// ---- GlobalTextList.TcGTLO
TEXTLIST GlobalTextList
  577 = ''
  578 = '%.1f'
  1916 = '%.1f '
  272 = '%.1f s'
  1255 = '%.2f'
  522 = '%.2f '
  324 = '%d'
  534 = '%i'
  168 = '%s'
  467 = '+'
  2312 = '+/-%.1f '
  462 = '+/-%.2f '
  1236 = '+/-%.f '
  759 = '-'
  43 = '1. Ben chặn hũ trên (s)' | vn: '1. Ben chặn hũ trên (s)' | eng: '1. Upper cylinder blocks jar (s)'
  1848 = '1. Ben dập nắp' | vn: '1. Ben dập nắp' | eng: '1. Cylinder presses lid'
  610 = '1. Ben dập nắp (s)' | vn: '1. Ben dập nắp (s)' | eng: '1. Cylinder presses lid (s)'
  2468 = '1. Ben hút, thả nắp' | vn: '1. Ben hút, thả nắp' | eng: '1. Cylinder sucks/release lid'
  1761 = '1. Ben hút/thả nắp (s)' | vn: '1. Ben hút/thả nắp (s)' | eng: '1. Cylinder sucks/release lid (s)'
  1520 = '1. Ben lược vào/ra' | vn: '1. Ben lược vào/ra' | eng: '1. Comb cylinder moves in/out'
  194 = '1. Ben lược vào/ra (s)' | vn: '1. Ben lược vào/ra (s)' | eng: '1. Comb cylinder moves in/out (s)'
  2358 = '1. Motor đảo thức ăn (Hz)' | vn: '1. Động cơ đảo thức ăn (Hz)' | eng: '1. Food Agitator motor (Hz)'
  2242 = '1. Phễu rung (Hz)' | vn: '1. Phễu rung (Hz)' | eng: '1. Vibrating funnel (Hz)'
  1784 = '1. Thời gian cân sâu (s)' | vn: '1. Thời gian cân sâu (s)' | eng: '1. Time for weighting larvae (s)'
  368 = '1. Thời gian cân thức ăn (s)' | vn: '1. Thời gian cân thức ăn (s)' | eng: '1. Time for weighting food (s)'
  621 = '1.Ben chặn hũ trên' | vn: '1. Ben chặn hũ trên' | eng: '1. The upper cylinder blocks the jar'
  1429 = '1.Khối lượng (g)' | vn: '1. Khối lượng (g)' | eng: '1. The mass (g)'
  758 = '1.Khối lượng yêu cầu (g)' | vn: '1. Khối lượng yêu cầu (g)' | eng: '1. The desire mass (g)'
  1103 = '1.Số Shoot' | vn: '1. Số Shoot' | eng: '1. Shoot number'
  1518 = '1/2'
  870 = '10. Khoảng trễ (s)' | vn: '10. Khoảng trễ (s)' | eng: '10. Delay (s)'
  2444 = '11. Tốc độ băng tải đầu ra (Hz)' | vn: '11. Tốc độ băng tải đầu ra (Hz)' | eng: '11. Speed of output conveyor (Hz)'
  3265 = '11. Tốc độ đảo thức ăn (Hz)' | vn: '11. Tốc độ đảo thức ăn (Hz)' | eng: '11. Speed of agitator motor (Hz)'
  3571 = '11. Tốc độ động cơ đảo (Hz)' | vn: '11. Tốc độ động cơ đảo (Hz)' | eng: '11. Speed of agitator motor (Hz)'
  254 = '2. Ben chặn hũ dưới (s)' | vn: '2. Ben chặn hũ dưới (s)' | eng: '2. Lower cylinder blocks jar (s)'
  85 = '2. Ben chặn nắp (s)' | vn: '2. Ben chặn nắp (s)' | eng: '2. Cylinder blocks lid (s)'
  2129 = '2. Ben chặn nắp trên ray' | vn: '2. Ben chặn nắp trên ray' | eng: '2. Cylinder blocks lid in rail'
  4542 = '2. Ben chặn sâu' | vn: '2. Ben chặn sâu ' | eng: '2. Cylinder blocks larvae'
  89 = '2. Ben di chuyển lược' | vn: '2. Ben di chuyển lược' | eng: '2. Cylinder moves comb'
  1937 = '2. Ben kẹp hũ (s)' | vn: '2. Ben kẹp hũ (s)' | eng: '2. Cylinder clamp jar (s)'
  1481 = '2. Khoảng trễ ben dập nắp rút về (s)' | vn: '2. Thời gian ben dập nắp rút về (s)' | eng: '2. Time for cylinder pressing lid retract (s)'
  204 = '2. Motor chia thức ăn (rpm)' | vn: '2. Động cơ chia thức ăn (rpm)' | eng: '2. Food dispenser motor (rpm)'
  588 = '2. Sai số (%)' | vn: '2. Sai số (%)' | eng: '2. Deviation (%)'
  863 = '2. Sai số cho phép (%)' | vn: '2. Sai số cho phép (%)' | eng: '2. Allowable deviation (%)'
  4394 = '2. Thời gian ben dập nắp rút về (s)' | vn: '2. Thời gian ben dập nắp rút về (s)' | eng: '2. Time for cylinder pressing lid retract (s)'
  2355 = '2. Thời gian ổn định hũ sâu (s)' | vn: '2. Thời gian ổn định hũ sâu (s)' | eng: '2. Time to stabilize the larvae jar (s)'
  4032 = '2. Thời gian ổn định hũ thức ăn (s)' | vn: '2. Thời gian ổn định hũ thức ăn (s)' | eng: '2. Time to stabilize the food jar (s)'
  311 = '2.Ben chặn hũ dưới' | vn: '2. Ben chặn hũ dưới' | eng: '2. The lower cylinder blocks the jar'
  3026 = '2/2'
  98 = '3. Ben chặn sâu (s)' | vn: '3. Ben chặn sâu (s)' | eng: '3. Cylinder blocks larvae (s)'
  198 = '3. Ben di chuyển lược (s)' | vn: '3. Ben di chuyển lược (s)' | eng: '3. Cylinder moves comb (s)'
  1881 = '3. Ben kẹp hũ, đối diện lược' | vn: '3. Ben kẹp hũ, đối diện lược' | eng: '3. Cylinder clamp the jar (s)'
  779 = '3. Kiểm tra hết hũ (s)' | vn: '3. Kiểm tra hết hũ (s)' | eng: '3. The jar is getting low (s)'
  1590 = '3. Kiểm tra hết nắp (s)' | vn: '3. Kiểm tra hết nắp (s)' | eng: '3. The lid is getting low (s)'
  1960 = '3. Thời gian đảo chiều động cơ trộn thức ăn (s)' | vn: '3. Thời gian đảo chiều động cơ trộn thức ăn (s)' | eng: '3. Timer for reversing agitator motor (s)'
  952 = '3. Tốc độ cấp I (Hz)' | vn: '3. Tốc độ cấp I (Hz)' | eng: '3. The velocity (Hz)'
  455 = '3. Tốc độ cấp I (rpm)' | vn: '3. Tốc độ cấp I (rpm)' | eng: '3. The velocity I (rpm)'
  3651 = '3. Tốc độ I (Hz)' | vn: '3. Tốc độ I (Hz)' | eng: '3. The velocity I (Hz)'
  1182 = '3. Tốc độ I (rpm)' | vn: '3. Tốc độ I (rpm)' | eng: '3. The velocity I (rpm)'
  3921 = '3. Van hút nắp' | vn: '3. Van hút nắp' | eng: '3. Valve sucks lid '
  740 = '3.Ben hút/thả hũ' | vn: '3. Ben hút/thả hũ' | eng: '3. Cylinder sucks/release jar'
  594 = '4. Kiểm tra hút được nắp (s)' | vn: '4. Kiểm tra hút được nắp (s)' | eng: '4. The lid is suctioned (s)'
  413 = '4. Kiểm tra hết sâu (s)' | vn: '4. Kiểm tra hết sâu (s)' | eng: '4. Check running out of larvae (s)'
  1166 = '4. Kiểm tra kẹt hũ (s)' | vn: '4. Kiểm tra kẹt hũ (s)' | eng: '4. The jar is stucked (s)'
  118 = '4. Thời gian đảo chiều động cơ chia thức ăn (s)' | vn: '4. Thời gian đảo chiều động cơ chia thức ăn (s)' | eng: '4. Timer for reversing (s)'
  4404 = '4. Tốc độ cấp II (Hz)' | vn: '4. Tốc độ cấp II (Hz)' | eng: '4. The velocity I (Hz)'
  297 = '4. Tốc độ cấp II (rpm)' | vn: '4. Tốc độ cấp II (rpm)' | eng: '4. The velocity II (rpm)'
  1764 = '4. Tốc độ II (Hz)' | vn: '4. Tốc độ II (Hz)' | eng: '4. The velocity II (Hz)'
  344 = '4. Tốc độ II (rpm)' | vn: '4. Tốc độ II (rpm)' | eng: '4. The velocity II (rpm)'
  86 = '4. Van hút định vị hũ' | vn: '4. Van hút định vị hũ' | eng: '4. Suction valve locates the jar'
  2844 = '5. Ben chặn hũ trên đẩy ra (s)' | vn: '5. Ben chặn hũ trên đẩy ra (s)' | eng: '5. Upper clinder blocks jar extend (s)'
  2498 = '5. Kiểm tra hết thức ăn (s)' | vn: '5, Kiểm tra hết thức ăn (s)' | eng: '5. Check running out of food (s)'
  2430 = '5. Ngắt hút (s)' | vn: '5. Ngắt hút (s)' | eng: '5. Shut off suction (s)'
  3883 = '5. Tốc độ cấp III (Hz)' | vn: '5. Tốc độ cấp III (Hz)' | eng: '5. The velocity III (Hz)'
  1037 = '5. Tốc độ cấp III (rpm)' | vn: '5. Tốc độ cấp III (rpm)' | eng: '5. The velocity III (rpm)'
  4207 = '5. Tốc độ III (Hz)' | vn: '5. Tốc độ III (Hz)' | eng: '5. The velocity III (Hz)'
  353 = '5. Tốc độ III (rpm)' | vn: '5. Tốc độ III (rpm)' | eng: '5. The velocity III (rpm)'
  2962 = '6. Ben hút/thả hũ (s)' | vn: '6. Ben hút/thả hũ (s)' | eng: '6. Cylinder sucks/releases jar (s)'
  2859 = '6. Ben hút/thả hũ(s)' | vn: '6. Ben hút/thả hũ (s)' | eng: '6. Cylinder sucks/releases jar (s)'
  657 = '6. Chuyển I - II (%)' | vn: '6. Chuyển I - II (%)' | eng: '6. Change I - II (%)'
  18 = '6. Vị trí chuyển cấp I - II (%)' | vn: '6. Vị trí chuyển cấp I - II (%)' | eng: '6. Postion change speed I - II (%)'
  1654 = '7. Ben hút/thả hũ rút về (s)' | vn: '7. Ben hút/thả hũ rút về (s)' | eng: '7. Cylinder sucks/releases jar retract (s)'
  865 = '7. Chuyển II - III (%)' | vn: '7. Chuyển II - III (%)' | eng: '7. Change II - III (%)'
  564 = '7. Vị trí chuyển cấp II - III (%)' | vn: '7. Vị trí chuyển cấp II - III (%)' | eng: '7. Position change speed II - III (%)'
  965 = '8. Ngắt hút (s)' | vn: '8. Ngắt hút (s)' | eng: '8. Stop suction (s)'
  677 = '8. Tải trọng tối đa (g)' | vn: '8. Tải trọng tối đa (g)' | eng: '8. Maximum payload (g)'
  1330 = '9. Vị trí dừng (%)' | vn: '9. Vị trí dừng (%)' | eng: '9. Halt position (%)'
  1341 = '9.Kích hút (s)' | vn: '9. Kích hút (s)' | eng: '9. Suction (s)'
  2827 = 'Bypass cửa' | vn: 'Bypass cửa' | eng: 'Bypass door'
  1689 = 'Bypass Nắp' | vn: 'Bypass Nắp' | eng: 'Bypass lid'
  1003 = 'Bypass Sâu' | vn: 'Bypass Sâu' | eng: 'Bypass larvae'
  207 = 'Bypass Thức ăn' | vn: 'Bypass Thức ăn' | eng: 'Bypass food'
  642 = 'Bạn có muốn xóa không?' | vn: 'Bạn có muốn xóa không?' | eng: 'Do you want to delete?'
  917 = 'Chạy' | vn: 'Chạy' | eng: 'Run'
  137 = 'Clear' | vn: 'Xóa' | eng: 'Clear'
  352 = 'Cài đặt' | vn: 'Cài đặt' | eng: 'Setting'
  503 = 'Có' | vn: 'Có' | eng: 'Yes'
  689 = 'Cụm cân sâu' | vn: 'Cụm cân sâu' | eng: 'Weighing larvae'
  775 = 'Cụm cấp hũ' | vn: 'Cụm cấp hũ' | eng: 'Jar supply'
  129 = 'Cụm cấp nắp' | vn: 'Cụm cấp nắp' | eng: 'Lid supply'
  838 = 'Cụm cấp thức ăn' | vn: 'Cụm cấp thức ăn' | eng: 'Food supply'
  454 = 'Cụm dập nắp' | vn: 'Cụm dập nắp' | eng: 'Pressing lid'
  80 = 'Cụm transfer' | vn: 'Cụm transfer' | eng: 'Transfer'
  1210 = 'DELAY LINE 1' | vn: 'THỜI GIAN TRẠM 1' | eng: 'TIMER LINE 1'
  1442 = 'DELAY LINE 2' | vn: 'THỜI GIAN TRẠM 2' | eng: 'TIMER LINE 2'
  61 = 'Describe'
  236 = 'Dừng' | vn: 'Dừng' | eng: 'Stop'
  643 = 'Dừng hút' | vn: 'Dừng hút' | eng: 'Stop suction'
  781 = 'Engineer'
  196 = 'Hút' | vn: 'Hút' | eng: 'Suck'
  2112 = 'Hết ca' | vn: 'Hết ca' | eng: 'End shift'
  1181 = 'ID' | vn: 'ID' | eng: 'ID'
  836 = 'INPUT' | vn: 'NGÕ VÀO' | eng: 'INPUT'
  184 = 'Không' | vn: 'Không' | eng: 'No'
  640 = 'Khối lượng cốc (g)' | vn: 'Khối lượng cốc (g)' | eng: 'Mass of cup (g)'
  523 = 'Khối lượng sâu (g)' | vn: 'Khối lượng sâu (g)' | eng: 'Mass of larvae (g)'
  474 = 'Khối lượng thức ăn (g)' | vn: 'Khối lượng thức ăn (g)' | eng: 'Mass of food (g)'
  1680 = 'LINE 1' | vn: 'TRẠM 1' | eng: 'LINE 1'
  1088 = 'LINE 2' | vn: 'TRẠM 2' | eng: 'LINE 2'
  849 = 'Lưu' | vn: 'Lưu' | eng: 'Save'
  1378 = 'Lựa chọn của bạn' | vn: 'Lựa chọn của bạn' | eng: 'Your choice'
  257 = 'MÀN HÌNH CHÍNH LINE 1' | vn: 'MÀN HÌNH CHÍNH TRẠM 1' | eng: 'MAIN LINE 1 SCREEN'
  4 = 'MÀN HÌNH CHÍNH LINE 2' | vn: 'MÀN HÌNH CHÍNH TRẠM 2' | eng: 'MAIN LINE 2 SCREEN'
  1168 = 'MÀN HÌNH CHẠY TAY LINE 1' | vn: 'MÀN HÌNH CHẠY TAY TRẠM 1' | eng: 'MANUAL LINE 1 SCREEN'
  762 = 'MÀN HÌNH CHẠY TAY LINE 2' | vn: 'MÀN HÌNH CHẠY TAY TRẠM 2' | eng: 'MANUAL LINE 2 SCREEN'
  1368 = 'MÀN HÌNH CÀI KHOẢNG TRỄ LINE 1' | vn: 'MÀN HÌNH CÀI KHOẢNG TRỄ TRẠM 1' | eng: 'SETTING DELAYS LINE 1'
  1237 = 'MÀN HÌNH CÀI KHOẢNG TRỄ LINE 2' | vn: 'MÀN HÌNH CÀI KHOẢNG TRỄ TRẠM 2' | eng: 'SETTING DELAYS LINE 2'
  386 = 'MÀN HÌNH CÀI ĐẶT LINE 1' | vn: 'MÀN HÌNH CÀI ĐẶT TRẠM 1' | eng: 'SETTINGS LINE 1 SCREEN'
  1892 = 'MÀN HÌNH CÀI ĐẶT LINE 2' | vn: 'MÀN HÌNH CÀI ĐẶT TRẠM 2' | eng: 'SETTINGS LINE 2 SCREEN'
  786 = 'MÀN HÌNH IO LINE 1' | vn: 'MÀN HÌNH IO TRẠM 1' | eng: 'IO LINE 1 SCREEN'
  798 = 'MÀN HÌNH IO LINE 2' | vn: 'MÀN HÌNH IO TRẠM 2' | eng: 'IO LINE 2 SCREEN'
  833 = 'MÀN HÌNH LƯU THÔNG SỐ LINE 1' | vn: 'MÀN HÌNH LƯU THÔNG SỐ TRẠM 1' | eng: 'PARAMETERS STORAGE LINE 1'
  1067 = 'MÀN HÌNH LƯU THÔNG SỐ LINE 2' | vn: 'MÀN HÌNH LƯU THÔNG SỐ TRẠM 2' | eng: 'PARAMETERS STORAGE LINE 2'
  4017 = 'MÀN HÌNH LỖI TRẠM 1' | vn: 'MÀN HÌNH LỖI TRẠM 1' | eng: 'ALARM SCREEN LINE 1'
  1028 = 'MÀN HÌNH LỖI TRẠM 2' | vn: 'MÀN HÌNH LỖI TRẠM 2' | eng: 'ALARM SCREEN LINE 2'
  1780 = 'MÀN HÌNH THÔNG SỐ TRẠM 1' | vn: 'MÀN HÌNH THÔNG SỐ TRẠM 1' | eng: 'PARAMETERS SCREEN LINE 1'
  1857 = 'MÀN HÌNH THÔNG SỐ TRẠM 2' | vn: 'MÀN HÌNH THÔNG SỐ TRẠM 2' | eng: 'PARAMETERS SCREEN LINE 2'
  1188 = 'Mô tả' | vn: 'Mô tả' | eng: 'Description'
  1449 = 'Ngược' | vn: 'Ngược' | eng: 'Reverse'
  777 = 'None'
  1079 = 'Năng suất (cup/h)' | vn: 'Năng suất(cốc/h)\t\t' | eng: 'Product(cup/h)'
  669 = 'Nạp' | vn: 'Nạp' | eng: 'Load'
  784 = 'Operator'
  219 = 'OUTPUT' | vn: 'NGÕ RA' | eng: 'OUTPUT'
  1453 = 'PARAMETER' | vn: 'THÔNG SỐ' | eng: 'PARAMETER'
  886 = 'Rút về' | vn: 'Rút về' | eng: 'Retract'
  139 = 'Sai số sâu (%)' | vn: 'Sai số sâu (%)' | eng: 'Deviation of larvae (%)'
  625 = 'Sai số thức ăn (%)' | vn: 'Sai số thức ăn (%)' | eng: 'Deviation of food (%)'
  478 = 'START' | vn: 'Bắt đầu' | eng: 'Start'
  3882 = 'Start page' | vn: 'Start page' | eng: 'Start page'
  440 = 'Status'
  12 = 'STOP' | vn: 'Dừng' | eng: 'Stop'
  62 = 'Sâu' | vn: 'Sâu' | eng: 'Larva'
  587 = 'SÂU' | vn: 'Sâu' | eng: 'Larva'
  909 = 'TG cân sâu' | vn: 'TG cân sâu' | eng: 'Time of weight larvae'
  2214 = 'TG cân thức ăn' | vn: 'TG cân thức ăn' | eng: 'Time of weight food'
  2059 = 'Thuận' | vn: 'Thuận' | eng: 'Forward'
  1204 = 'Thời gian' | vn: 'Thời gian' | eng: 'Time'
  1876 = 'Thời gian (s)' | vn: 'Thời gian (s)' | eng: 'Time (s)'
  294 = 'Thức ăn' | vn: 'Thức ăn' | eng: 'Food'
  513 = 'THỨC ĂN' | vn: 'Thức ăn' | eng: 'Food'
  877 = 'Thực tế' | vn: 'Thực tế' | eng: 'Actual'
  48 = 'Time'
  1196 = 'Trạng thái' | vn: 'Trạng thái' | eng: 'Status'
  771 = 'Trạng thái hoạt động' | vn: 'Trạng thái hoạt động' | eng: 'Operation status'
  1711 = 'Trộn' | vn: 'Trộn' | eng: 'Mix'
  2142 = 'Tạm dừng' | vn: 'Tạm dừng' | eng: 'Pause'
  2305 = 'Tốc độ (g/s)' | vn: 'Tốc độ (g/s)' | eng: 'Velocity (g/s)'
  754 = 'Tổng khối lượng (g)' | vn: 'Tổng khối lượng (g)' | eng: 'Mass total (g)'
  1399 = 'Tổng số cốc đã cân' | vn: 'Tổng số cốc đã cân' | eng: 'Total cups weighted'
  1621 = 'U1I1-1. Nút Start' | vn: 'U1I1-1. Nút Start' | eng: 'U1I1-1. Start button'
  3076 = 'U1I1-2. Nút Stop' | vn: 'U1I1-2. Nút Stop' | eng: 'U1I1-2. Stop button'
  536 = 'U1I1-3. Nút Reset' | vn: 'U1I1-3. Nút Reset' | eng: 'U1I1-3. Rest button'
  3249 = 'U1I2-4. Cảm biến báo thiếu hũ' | vn: 'U1I2-4. Cảm biến báo thiếu hũ' | eng: 'U1I2-4. Sensor detecting jar is getting low'
  2058 = 'U1I2-5. Cảm biến rút về của ben chặn hũ trên' | vn: 'U1I2-5. Cảm biến rút về của ben chặn hũ trên' | eng: 'U1I2-5. Retract sensor of upper cylinder'
  1695 = 'U1I2-6. Cảm biến rút về của ben chặn hũ dưới' | vn: 'U1I2-6. Cảm biến rút về của ben chặn hũ dưới' | eng: 'U1I2-6. Retract sensor of lower cylinder'
  3389 = 'U1I2-7. Cảm biến đẩy ra của ben chặn hũ dưới' | vn: 'U1I2-7. Cảm biến đẩy ra của ben chặn hũ dưới' | eng: 'U1I2-7. Extend sensor of upper cylinder'
  71 = 'U1I2-8. Cảm biến báo kẹt hũ' | vn: 'U1I2-8. Cảm biến báo kẹt hũ' | eng: 'U1I2-8. Sensor detecting jar is stucked'
  4241 = 'U1I3-1. Cảm biến rút về ben chặn sâu' | vn: 'U1I3-1. Cảm biến rút về ben chặn sâu' | eng: 'U1I3-1. Retract sensor of cylinder blocks larvae'
  500 = 'U1I3-2. Cảm biến báo thiếu nắp' | vn: 'U1I3-2. Cảm biến báo thiếu nắp' | eng: 'U1I3-2. Sensor detecting lid is getting low'
  1849 = 'U1I3-3. Cảm biến rút về của ben chặn nắp' | vn: 'U1I3-3. Cảm biến rút về của ben chặn nắp' | eng: 'U1I3-3. Retract sensor of cylinder blocks lid'
  31 = 'U1I3-4. Cảm biến đẩy ra của ben chặn nắp' | vn: 'U1I3-4. Cảm biến đẩy ra của ben chặn nắp' | eng: 'U1I3-4. Extend sensor of cylinder blocks lid'
  277 = 'U1I3-5. Cảm biến trên của ben hút nắp' | vn: 'U1I3-5. Cảm biến trên của ben hút nắp' | eng: 'U1I3-5. Upper sensor of cylinder sucks lid'
  2845 = 'U1I3-6. Cảm biến dưới của ben hút nắp ' | vn: 'U1I3-6. Cảm biến dưới của ben hút nắp' | eng: 'U1I3-6. Lower sensor of cylinder sucks lid'
  2605 = 'U1I3-7. Cảm biến báo hút được nắp' | vn: 'U1I3-7. Cảm biến báo hút được nắp' | eng: 'U1I3-7. Sensor detecting lid is sucked'
  3955 = 'U1I3-8. Cảm biến trên của ben dập nắp' | vn: 'U1I3-8. Cảm biến trên của ben dập nắp' | eng: 'U1I3-8. Upper sensor of cylinder presses lid'
  3907 = 'U1I4-1. Cảm biến dưới của ben dập nắp' | vn: 'U1I4-1. Cảm biến dưới của ben dập nắp' | eng: 'U1I4-1. Lower sensor of cylinder presses lid'
  876 = 'U1I4-2. Cảm biến rút về của ben lược' | vn: 'U1I4-2. Cảm biến rút về của ben lược' | eng: 'U1I4-2. Retract sensor of comb cylinder'
  2630 = 'U1I4-3. Cảm biến đẩy ra của ben lược' | vn: 'U1I4-3. Cảm biến đẩy ra của ben lược' | eng: 'U1I4-3. Extend sensor of comb cylinder'
  4377 = 'U1I4-4. Cảm biến rút về của ben di chuyển lược' | vn: 'U1I4-4. Cảm biến rút về của ben di chuyển lược' | eng: 'U1I4-4. Retract sensor of cylinder moves comb'
  2666 = 'U1I4-5. Cảm biến đẩy ra của ben di chuyển lược' | vn: 'U1I4-5. Cảm biến đẩy ra của ben di chuyển lược' | eng: 'U1I4-5. Extend sensor of cylidner moves comb'
  1344 = 'U1I4-6. Cảm biến rút về của ben kẹp hũ ' | vn: 'U1I4-6. Cảm biến rút về của ben kẹp hũ' | eng: 'U1I4-6. Retract sensor of cylinder clamp jar'
  1519 = 'U1I4-7. Cảm biến đẩy ra của ben kẹp hũ ' | vn: 'U1I4-7. Cảm biến đẩy ra của ben kẹp hũ' | eng: 'U1I4-7. Extend sensor of cylinder clamp jar'
  1627 = 'U1I4-8. Cảm biến phát hiện hũ ở chỗ cân thức ăn' | vn: 'U1I4-8. Cảm biến phát hiện hũ ở chỗ cân thức ăn' | eng: 'U1I4-8. Sensor detecting jar in food station'
  3159 = 'U1I5-1. Cảm biến phát hiện hũ ở chỗ cân sâu' | vn: 'U1I5-1. Cảm biến phát hiện hũ ở chỗ cân sâu' | eng: 'U1I5-1. Sensor detecting jar in larvae station'
  524 = 'U1I5-2. Cảm biến báo thiếu hũ' | vn: 'U1I5-2. Cảm biến báo thiếu hũ' | eng: 'U1I5-2. Sensor detecting jar is getting low'
  2400 = 'U1I5-3. Cảm biến rút về của ben chặn hũ trên' | vn: 'U1I5-3. Cảm biến rút về của ben chặn hũ trên' | eng: 'U1I5-3. Retract sensor of upper cylinder'
  2538 = 'U1I5-4. Cảm biến rút về của ben chặn hũ dưới' | vn: 'U1I5-4. Cảm biến rút về của ben chặn hũ dưới' | eng: 'U1I5-4. Retract sensor of lower cylinder'
  177 = 'U1I5-5. Cảm biến đẩy ra của ben chặn hũ dưới' | vn: 'U1I5-5. Cảm biến đẩy ra của ben chặn hũ dưới' | eng: 'U1I5-5. Extend sensor of lower cylinder'
  2643 = 'U1I5-6. Cảm biến báo kẹt hũ' | vn: 'U1I5-6. Cảm biến báo kẹt hũ' | eng: 'U1I5-6. Sensor detecting jar is stucked'
  1877 = 'U1I5-7. Cảm biến rút về ben chặn sâu' | vn: 'U1I5-7. Cảm biến rút về ben chặn sâu' | eng: 'U1I5-7. Retract sensor of cylinder blocks larvae'
  2706 = 'U1I5-8. Cảm biến báo thiếu nắp' | vn: 'U1I5-8. Cảm biến báo thiếu nắp' | eng: 'U1I5-8. Sensor detecting lid is getting low'
  3822 = 'U1I6-1. Cảm biến rút về của ben chặn nắp' | vn: 'U1I6-1. Cảm biến rút về của ben chặn nắp' | eng: 'U1I6-1. Retract sensor of cylinder blocks lid'
  2003 = 'U1I6-2. Cảm biến đẩy ra của ben chặn nắp' | vn: 'U1I6-2. Cảm biến đẩy ra của ben chặn nắp' | eng: 'U1I6-2. Extend sensor of cylinder blocks lid'
  787 = 'U1I6-3. Cảm biến trên của ben hút nắp' | vn: 'U1I6-3. Cảm biến trên của ben hút nắp' | eng: 'U1I6-3. Upper sensor of cylinder sucks lid'
  1106 = 'U1I6-4. Cảm biến dưới của ben hút nắp ' | vn: 'U1I6-4. Cảm biến dưới của ben hút nắp' | eng: 'U1I6-4. Lower sensor of cylinder sucks lid'
  2433 = 'U1I6-5. Cảm biến báo hút được nắp' | vn: 'U1I6-5. Cảm biến báo hút được nắp' | eng: 'U1I6-5. Sensor detecting lid is sucked'
  2961 = 'U1I6-6. Cảm biến trên của ben dập nắp' | vn: 'U1I6-6. Cảm biến trên của ben dập nắp' | eng: 'U1I6-6. Upper sensor of cylinder presses lid'
  397 = 'U1I6-7. Cảm biến dưới của ben dập nắp' | vn: 'U1I6-7. Cảm biến dưới của ben dập nắp' | eng: 'U1I6-7. Lower sensor of cylinder presses lid'
  1052 = 'U1I6-8. Cảm biến rút về của ben lược' | vn: 'U1I6-8. Cảm biến rút về của ben lược' | eng: 'U1I6-8. Retract sensor of comb cylinder'
  4010 = 'U1I7-1. Cảm biến đẩy ra của ben lược' | vn: 'U1I7-1. Cảm biến đẩy ra của ben lược' | eng: 'U1I7-1. Extend sensor of comb cylinder'
  1534 = 'U1I7-10. Cảm biến cửa 3' | vn: 'U1I7-10. Cảm biến cửa 3' | eng: 'U1I7-10. Sensor door 3'
  550 = 'U1I7-10.Cảm biến cửa 3' | vn: 'U1I7-10. Cảm biến cửa 3' | eng: 'U1I7-10. Sensor door 3'
  1820 = 'U1I7-2. Cảm biến rút về của ben di chuyển lược' | vn: 'U1I7-2. Cảm biến rút về của ben di chuyển lược' | eng: 'U1I7-2. Retract sensor of cylinder moves comb'
  2657 = 'U1I7-3. Cảm biến đẩy ra của ben di chuyển lược' | vn: 'U1I7-3. Cảm biến đẩy ra của ben di chuyển lược' | eng: 'U1I7-3. Extend sensor of cylinder moves comb'
  360 = 'U1I7-4. Cảm biến rút về của ben kẹp hũ' | vn: 'U1I7-4. Cảm biến rút về của ben kẹp hũ' | eng: 'U1I7-4. Retract sensor of cylinder clamp jar'
  1051 = 'U1I7-5. Cảm biến đẩy ra của ben kẹp hũ' | vn: 'U1I7-5. Cảm biến đẩy ra của ben kẹp hũ' | eng: 'U1I7-5. Extend sensor of cylinder clamp jar'
  3158 = 'U1I7-6. Cảm biến phát hiện hũ ở chỗ cân thức ăn' | vn: 'U1I7-6. Cảm biến phát hiện hũ ở chỗ cân thức ăn' | eng: 'U1I7-6. Sensor detecting jar in food station'
  2876 = 'U1I7-7. Cảm biến phát hiện hũ ở chỗ cân sâu' | vn: 'U1I7-7. Cảm biến phát hiện hũ ở chỗ cân sâu' | eng: 'U1I7-7. Sensor detecting jar in larvae station'
  210 = 'U1I7-8. Cảm biến cửa 1' | vn: 'U1I7-8. Cảm biến cửa 1' | eng: 'U1I7-8. Sensor door 1'
  761 = 'U1I7-9. Cảm biến cửa 2' | vn: 'U1I7-9. Cảm biến cửa 2' | eng: 'U1I7-9. Sensor door 2'
  4190 = 'U1O1-1. Đèn báo chạy chế độ tự động' | vn: 'U1O1-1. Đèn báo chạy chế độ tự động' | eng: 'U1O1-1. Auto start lamp'
  1081 = 'U1O1-10. Động cơ chia thức ăn' | vn: 'U1O1-10. Động cơ chia thức ăn' | eng: 'U1O1-10. Food dispenser motor'
  4307 = 'U1O1-12. Động cơ chia thức ăn' | vn: 'U1O1-12. Động cơ chia thức ăn' | eng: 'U1O1-12. Food dispenser motor'
  3445 = 'U1O1-13. Ben chặn hũ trên' | vn: 'U1O1-13. Ben chặn hũ trên' | eng: 'U1O1-13. Upper cylinder blocks jar'
  1336 = 'U1O1-14. Ben chặn hũ dưới' | vn: 'U1O1-14. Ben chặn hũ dưới' | eng: 'U1O1-14. Lower cylinder bocks jar'
  3055 = 'U1O1-15. Ben chặn sâu' | vn: 'U1O1-15. Ben chặn sâu' | eng: 'U1O1-15. Cylinder blocks larvae'
  3097 = 'U1O1-16. Ben chặn nắp' | vn: 'U1O1-16. Ben chặn nắp' | eng: 'U1O1-16. Cylinder blocks lid'
  3203 = 'U1O1-2. Đèn báo dừng chế độ tự động' | vn: 'U1O1-2. Đèn báo dừng chế độ tự động' | eng: 'U1O1-2. Auto stop lamp'
  1531 = 'U1O1-3. Động cơ đảo thức ăn ' | vn: 'U1O1-3. Động cơ đảo thức ăn' | eng: 'U1O1-3. Food agitator motor'
  2964 = 'U1O1-4. Phễu rung' | vn: 'U1O1-4. Phễu rung' | eng: 'U1O1-4. Vibrating funnel'
  1779 = 'U1O1-5. Băng tải đầu ra' | vn: 'U1O1-5. Băng tải đầu ra' | eng: 'U1O1-5. Output conveyor'
  336 = 'U1O1-6. Động cơ đảo thức ăn' | vn: 'U1O1-6. Động cơ đảo thức ăn' | eng: 'U1O1-6. Food agitator motor'
  3124 = 'U1O1-7. Phễu rung' | vn: 'U1O1-7. Phễu rung' | eng: 'U1O1-7. Vibrating funnel'
  4277 = 'U1O1-8. Còi' | vn: 'U1O1-8. Còi' | eng: 'U1O1-8. Horn'
  1546 = 'U1O2-1. Ben hút/thả nắp' | vn: 'U1O2-1. Ben hút/thả nắp' | eng: 'U1O2-1. Cylinder sucks/releases lid'
  4439 = 'U1O2-10. Ben chặn sâu' | vn: 'U1O2-10. Ben chặn sâu' | eng: 'U1O2-10. Cylinder blocks larvae'
  1589 = 'U1O2-11. Ben chặn nắp' | vn: 'U1O2-11. Ben chặn nắp' | eng: 'U1O2-11. Cylinder blocks lid'
  2376 = 'U1O2-12. Ben hút/thả nắp' | vn: 'U1O2-12. Ben hút/thả nắp' | eng: 'U1O2-12. Cylinder sucks/releases lid'
  2070 = 'U1O2-13. Van hút nắp' | vn: 'U1O2-13. Van hút nắp' | eng: 'U1O2-13. Valve sucks lid'
  1647 = 'U1O2-14. Van hút hũ' | vn: 'U1O2-14. Van hút hũ' | eng: 'U1O2-14. Valve sucks jar'
  2017 = 'U1O2-15. Ben dập nắp' | vn: 'U1O2-15. Ben dập nắp' | eng: 'U1O2-15. Cylinder presses lid'
  305 = 'U1O2-16. Ben kẹp hũ' | vn: 'U1O2-16. Ben kẹp hũ' | eng: 'U1O2-16. Cylinder clamp jar'
  4049 = 'U1O2-2. Van hút nắp' | vn: 'U1O2-2. Van hút nắp' | eng: 'U1O2-2. Valve sucks lid'
  3916 = 'U1O2-3. Van hút hũ' | vn: 'U1O2-3. Van hút hũ' | eng: 'U1O2-3. Valve sucks jar'
  4107 = 'U1O2-4. Ben dập nắp' | vn: 'U1O2-4. Ben dập nắp' | eng: 'U1O2-4. Cylinder presses lid'
  2321 = 'U1O2-5. Ben kẹp hũ' | vn: 'U1O2-5. Ben kẹp hũ' | eng: 'U1O2-5. Cylinder clamp jar'
  4004 = 'U1O2-6. Ben lược ra/vào' | vn: 'U1O2-6. Ben lược ra/vào' | eng: 'U1O2-6. Comb cylinder moves in/out'
  371 = 'U1O2-7. Ben di chuyển lược' | vn: 'U1O2-7. Ben di chuyển lược' | eng: 'U1O2-7. Cylinder moves comb'
  2551 = 'U1O2-8. Ben chặn hũ trên' | vn: 'U1O2-8. Ben chặn hũ trên' | eng: 'U1O2-8. Upper cylinder blocks jar'
  2149 = 'U1O2-9. Ben chặn hũ dưới' | vn: 'U1O2-9. Ben chặn hũ dưới' | eng: 'U1O2-9. Lower cylinder blocks jar'
  2052 = 'U1O3-1. Ben lược ra/vào' | vn: 'U1O3-1. Ben lược ra/vào' | eng: 'U1O3-1. Comb clinder moves in/out'
  2598 = 'U1O3-2. Ben di chuyển lược' | vn: 'U1O3-2. Ben di chuyển lược' | eng: 'U1O3-2. Cylinder moves comb'
  126 = 'Vui lòng nhập tên của bạn' | vn: 'Vui lòng nhập tên của bạn' | eng: 'Please enter your name'
  2236 = 'WARNING: %s'
  26 = 'Welcome' | vn: 'Welcome' | eng: 'Welcome'
  3677 = 'X'
  286 = 'Xóa' | vn: 'Xóa' | eng: 'Delete'
  1430 = 'Xả sâu' | vn: 'Xả sâu' | eng: 'Flush larvae'
  1211 = 'Xả thức ăn' | vn: 'Xả thức ăn' | eng: 'Flush food'
  3643 = 'Đăng nhập' | vn: 'Đăng nhập' | eng: 'Login'
  1411 = 'Đẩy ra' | vn: 'Đẩy ra' | eng: 'Extend'
  831 = 'Đặt về 0' | vn: 'Đặt về 0' | eng: 'Set 0'
END_TEXTLIST

// ---- VISUs/Alarm/N_Alarm.TcVIS
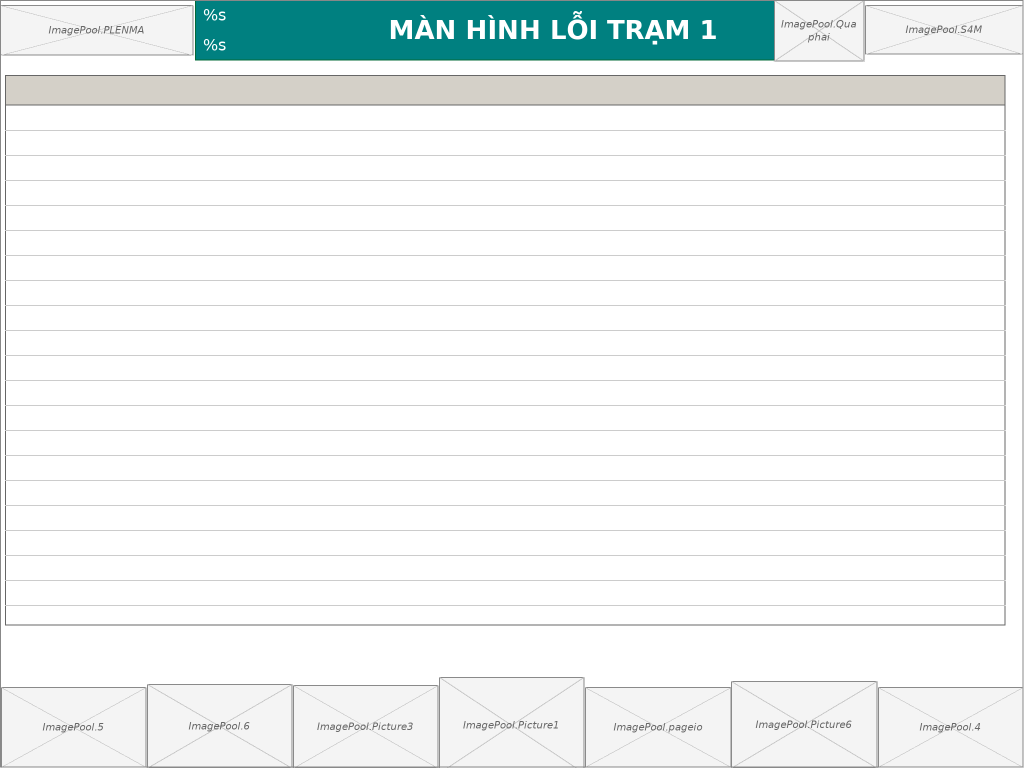
VISUALIZATION N_Alarm  // 1024x768
    Table (5,75 1000x550), invisible if: Not bVN, data array: AlarmList
        p3854506369: AlarmList[1,INDEX]
        p1892666644: AlarmList[2,INDEX]
        p338671338: AlarmList[3,INDEX]
        p2170511999: AlarmList[4,INDEX]
        p511219082: Mô tả
        p1755163831: Trạng thái
        p4092479075: Thời gian
    Table (5,75 1000x550), invisible if: bVN, data array: AlarmList3
        p3854506369: AlarmList3[1,INDEX]
        p1892666644: AlarmList3[2,INDEX]
        p338671338: AlarmList[3,INDEX]
        p2170511999: AlarmList[4,INDEX]
        p511219082: Describe
        p1755163831: Status
        p4092479075: Time
        p1791247317: AlarmList3[3,INDEX]
        p262371475: AlarmList3[4,INDEX]
    Frame (0,687 1024x80)
        shows N_Footer_Line1()
    Frame (0,0 1024x60)
        shows N_Header()
    Textfield (353,5 400x50), "MÀN HÌNH LỖI TRẠM 1"
    Image (774,0 90x61), image: ImagePool.Qua phai
        OnMouseClick: change screen: N_Alarm_1
END_VISUALIZATION

// ---- VISUs/Alarm/N_Alarm_1.TcVIS
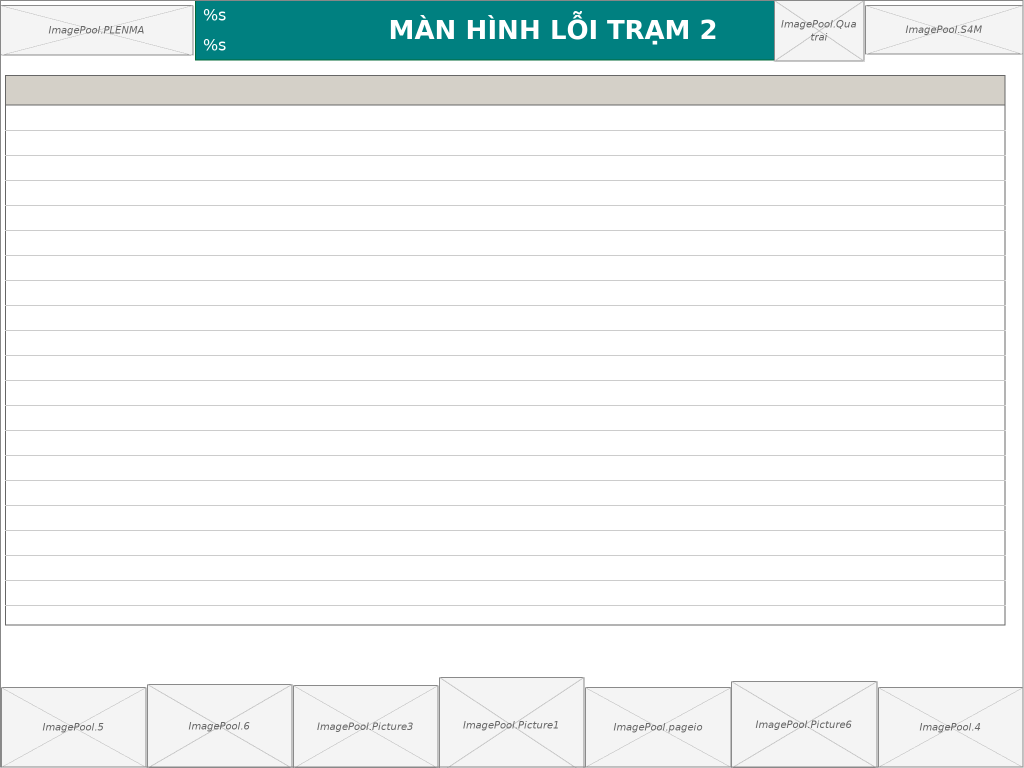
VISUALIZATION N_Alarm_1  // 1024x768
    Table (5,75 1000x550), invisible if: bVN, data array: AlarmList4
        p3854506369: AlarmList4[1,INDEX]
        p1892666644: AlarmList4[2,INDEX]
        p338671338: AlarmList[3,INDEX]
        p2170511999: AlarmList[4,INDEX]
        p511219082: Describe
        p1755163831: Status
        p4092479075: Time
        p1791247317: AlarmList4[3,INDEX]
        p262371475: AlarmList4[4,INDEX]
    Frame (0,687 1024x80)
        shows N_Footer_Line2()
    Frame (0,0 1024x60)
        shows N_Header()
    Textfield (353,5 400x50), "MÀN HÌNH LỖI TRẠM 2"
    Table (5,75 1000x550), invisible if: not bVN, data array: AlarmList2
        p3854506369: AlarmList2[1,INDEX]
        p1892666644: AlarmList2[2,INDEX]
        p338671338: AlarmList2[3,INDEX]
        p2170511999: AlarmList2[4,INDEX]
        p511219082: Mô tả
        p1755163831: Trạng thái
        p4092479075: Thời gian
    Image (774,0 90x61), image: ImagePool.Qua trai
        OnMouseClick: change screen: N_Alarm
END_VISUALIZATION

// ---- VISUs/IO/N_Parameter_1.TcVIS
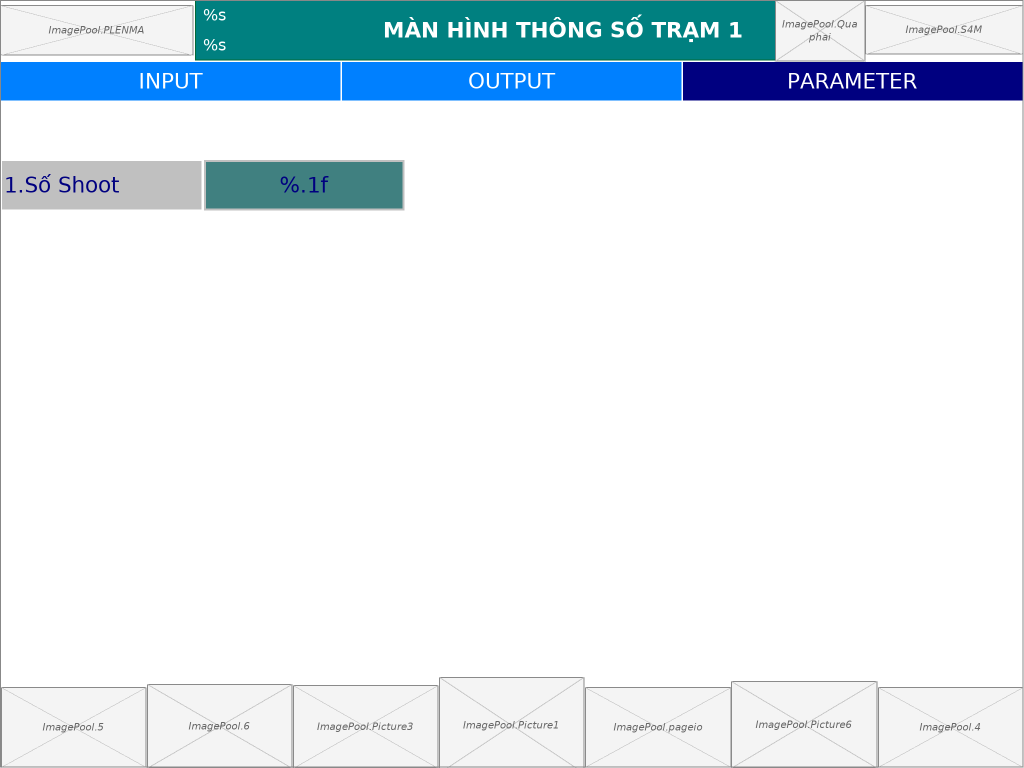
VISUALIZATION N_Parameter_1  // 1024x768
    Frame (0,0 1024x60)
        shows N_Header()
    Rectangle (0,61 341x40), "INPUT"
        OnMouseClick: change screen: N_PLC_I1
    Rectangle (341,61 341x40), "OUTPUT"
        OnMouseClick: change screen: N_PLC_O1
    Rectangle (682,61 341x40), "PARAMETER"
        OnMouseClick: change screen: N_Parameter_1
    Textfield (363,5 400x50), "MÀN HÌNH THÔNG SỐ TRẠM 1"
    Rectangle (1,160 201x50), "1.Số Shoot"
    Textfield (204,160 200x50), "%.1f", text variable: nShoot1
    Image (775,0 90x61), image: ImagePool.Qua phai
        OnMouseClick: change screen: N_Parameter_2
    Frame (0,687 1024x80)
        shows N_Footer_Line1()
END_VISUALIZATION

// ---- VISUs/IO/N_Parameter_2.TcVIS
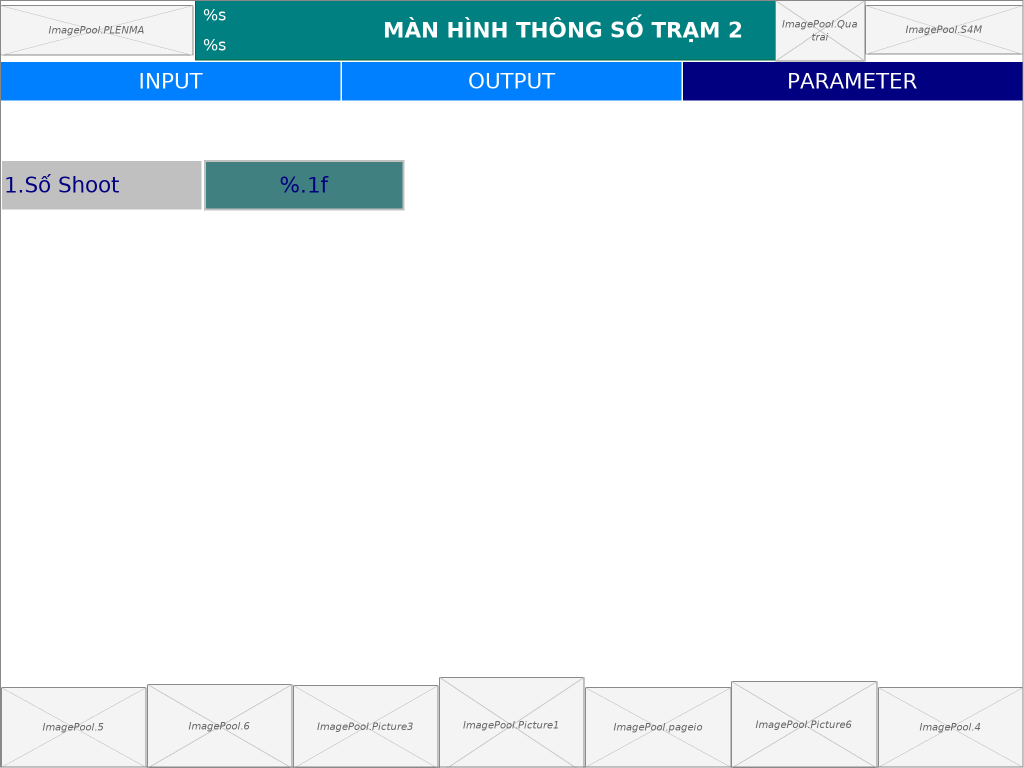
VISUALIZATION N_Parameter_2  // 1024x768
    Frame (0,0 1024x60)
        shows N_Header()
    Rectangle (0,61 341x40), "INPUT"
        OnMouseClick: change screen: N_PLC_I2
    Rectangle (341,61 341x40), "OUTPUT"
        OnMouseClick: change screen: N_PLC_O2
    Rectangle (682,61 341x40), "PARAMETER"
        OnMouseClick: change screen: N_Parameter_2
    Textfield (363,5 400x50), "MÀN HÌNH THÔNG SỐ TRẠM 2"
    Rectangle (1,160 201x50), "1.Số Shoot"
    Textfield (204,160 200x50), "%.1f", text variable: nShoot2
    Image (775,0 90x61), image: ImagePool.Qua trai
        OnMouseClick: change screen: N_Parameter_1
    Frame (0,687 1024x80)
        shows N_Footer_Line2()
END_VISUALIZATION

// ---- VISUs/IO/N_PLC_I1.TcVIS
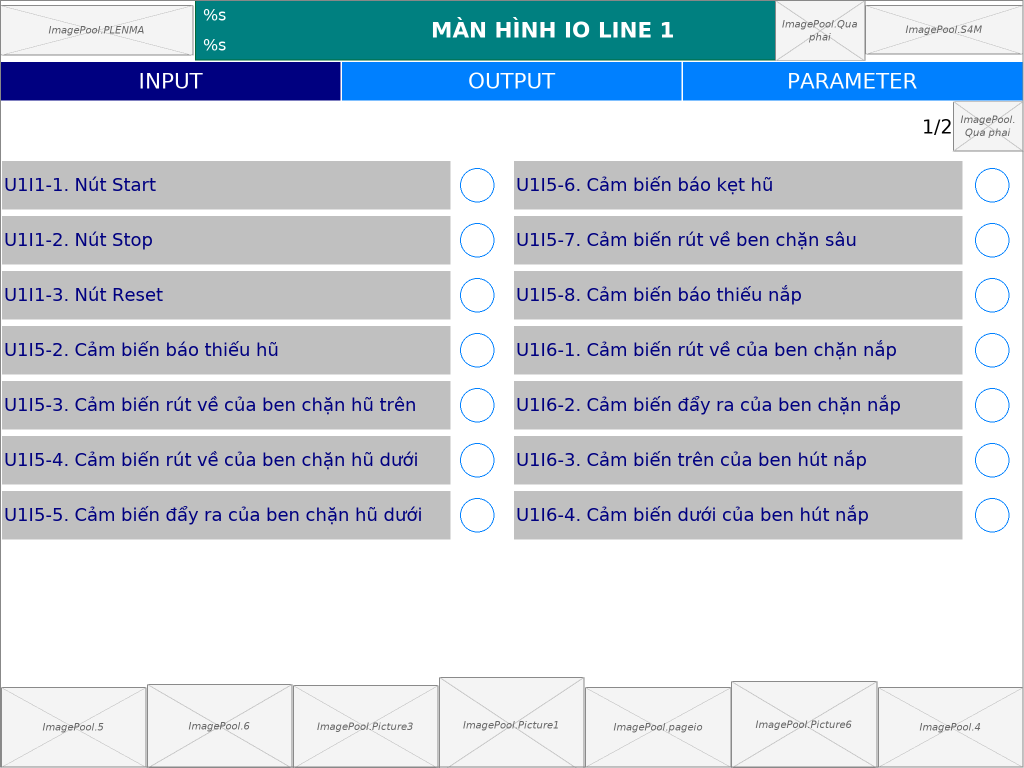
VISUALIZATION N_PLC_I1  // 1024x768
    Rectangle (886,102 103x50), "1/2"
    Frame (0,687 1024x80)
        shows N_Footer_Line1()
    Frame (0,0 1024x60)
        shows N_Header()
    Textfield (353,5 400x50), "MÀN HÌNH IO LINE 1"
    Image (775,0 90x61), image: ImagePool.Qua phai
        OnMouseClick: change screen: N_PLC_I2
    Rectangle (1,325 450x50), "U1I5-2. Cảm biến báo thiếu hũ"
    Rectangle (1,380 450x50), "U1I5-3. Cảm biến rút về của ben chặn hũ trên"
    Rectangle (1,435 450x50), "U1I5-4. Cảm biến rút về của ben chặn hũ dưới"
    Rectangle (1,490 450x50), "U1I5-5. Cảm biến đẩy ra của ben chặn hũ dưới"
    Rectangle (1,160 450x50), "U1I1-1. Nút Start"
    Rectangle (1,215 450x50), "U1I1-2. Nút Stop"
    Rectangle (1,270 450x50), "U1I1-3. Nút Reset"
    Ellipse (460,168 34x34), colour toggle: GVL_IO.bStart, input disabled if: true
    Ellipse (460,223 34x34), colour toggle: GVL_IO.bStop, input disabled if: true
    Ellipse (460,278 34x34), colour toggle: GVL_IO.bReset, input disabled if: true
    Ellipse (460,333 34x34), colour toggle: PR_Line01.fb_CupSupply.bCupEmpty, input disabled if: true
    Ellipse (460,388 34x34), colour toggle: PR_Line01.fb_CupSupply.fbCylinder_Up.bAtRetract, input disabled if: true
    Ellipse (460,443 34x34), colour toggle: PR_Line01.fb_CupSupply.fbCylinder_Dw.bAtRetract, input disabled if: true
    Ellipse (460,498 34x34), colour toggle: PR_Line01.fb_CupSupply.fbCylinder_Dw.bAtExtend, input disabled if: true
    Rectangle (513,490 450x50), "U1I6-4. Cảm biến dưới của ben hút nắp"
    Rectangle (513,160 450x50), "U1I5-6. Cảm biến báo kẹt hũ"
    Rectangle (513,215 450x50), "U1I5-7. Cảm biến rút về ben chặn sâu"
    Rectangle (513,270 450x50), "U1I5-8. Cảm biến báo thiếu nắp"
    Rectangle (513,325 450x50), "U1I6-1. Cảm biến rút về của ben chặn nắp"
    Rectangle (513,380 450x50), "U1I6-2. Cảm biến đẩy ra của ben chặn nắp"
    Rectangle (513,435 450x50), "U1I6-3. Cảm biến trên của ben hút nắp"
    Ellipse (975,168 34x34), colour toggle: PR_Line01.fb_CupSupply.bCupDrop, input disabled if: true
    Ellipse (975,498 34x34), colour toggle: PR_Line01.fb_LidSupply.fbCylinder_Suction.bAtExtend, input disabled if: true
        toggle GVL_OF_VU.bSensorOutOfLid[2]
    Ellipse (975,223 34x34), colour toggle: PR_Line01.fb_WormWeight.fbCylinder.bAtRetract, input disabled if: true
    Ellipse (975,278 34x34), colour toggle: PR_Line01.fb_LidSupply.bLidEmpty, input disabled if: true
    Ellipse (975,333 34x34), colour toggle: PR_Line01.fb_LidSupply.fbCylinder_LidStopper.bAtRetract, input disabled if: true
    Ellipse (975,388 34x34), colour toggle: PR_Line01.fb_LidSupply.fbCylinder_LidStopper.bAtExtend, input disabled if: true
    Ellipse (975,443 34x34), colour toggle: PR_Line01.fb_LidSupply.fbCylinder_Suction.bAtRetract, input disabled if: true
    Image (953,101 70x50), image: ImagePool.Qua phai
        OnMouseClick: change screen: N_PLC_I1_next
    Rectangle (341,61 341x40), "OUTPUT"
        OnMouseClick: change screen: N_PLC_O1
    Rectangle (0,61 341x40), "INPUT"
        OnMouseClick: change screen: N_PLC_I1
    Rectangle (682,61 341x40), "PARAMETER"
        OnMouseClick: change screen: N_Parameter_1
END_VISUALIZATION

// ---- VISUs/IO/N_PLC_I1_next.TcVIS
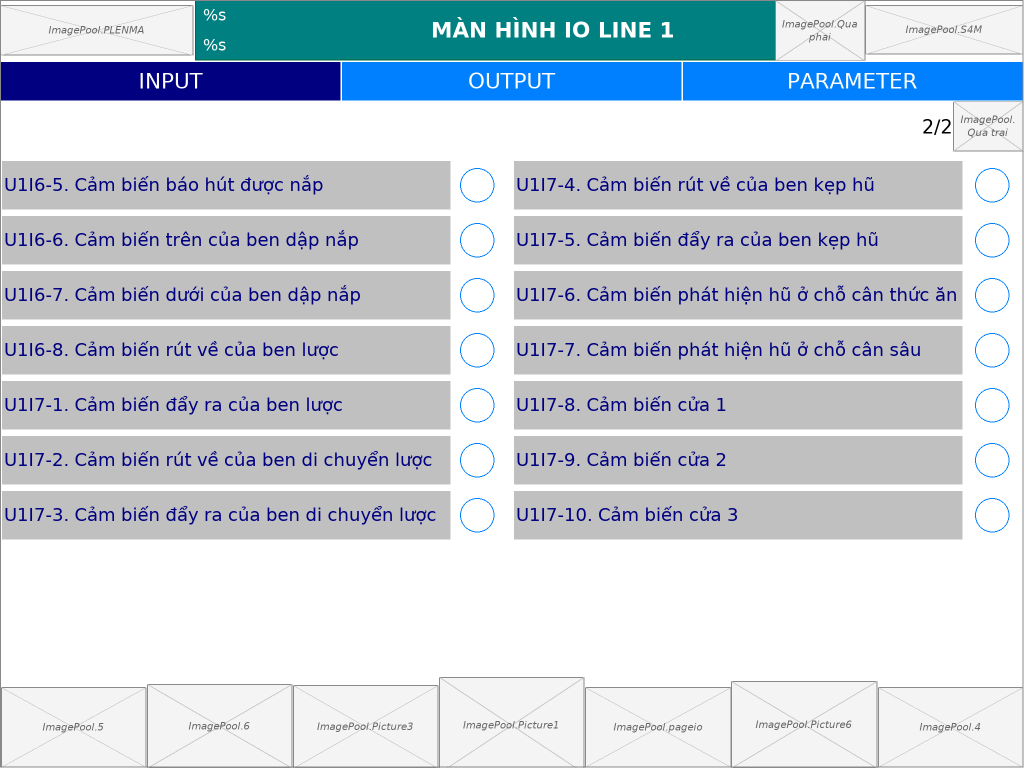
VISUALIZATION N_PLC_I1_next  // 1024x768
    Rectangle (886,102 103x50), "2/2"
    Frame (0,687 1024x80)
        shows N_Footer_Line1()
    Frame (0,0 1024x60)
        shows N_Header()
    Textfield (353,5 400x50), "MÀN HÌNH IO LINE 1"
    Image (775,0 90x61), image: ImagePool.Qua phai
        OnMouseClick: change screen: N_PLC_I2
    Rectangle (1,160 450x50), "U1I6-5. Cảm biến báo hút được nắp"
    Rectangle (1,215 450x50), "U1I6-6. Cảm biến trên của ben dập nắp"
    Rectangle (1,325 450x50), "U1I6-8. Cảm biến rút về của ben lược"
    Rectangle (1,270 450x50), "U1I6-7. Cảm biến dưới của ben dập nắp"
    Rectangle (1,380 450x50), "U1I7-1. Cảm biến đẩy ra của ben lược"
    Rectangle (1,435 450x50), "U1I7-2. Cảm biến rút về của ben di chuyển lược"
    Rectangle (1,490 450x50), "U1I7-3. Cảm biến đẩy ra của ben di chuyển lược"
    Ellipse (460,168 34x34), colour toggle: PR_Line01.fb_LidSupply.fbLidSuctionValve.bPressure, input disabled if: true
    Ellipse (460,223 34x34), colour toggle: PR_Line01.fb_LidClose.fbCylinder_LidClose.bAtRetract, input disabled if: true
    Ellipse (460,278 34x34), colour toggle: PR_Line01.fb_LidClose.fbCylinder_LidClose.bAtExtend, input disabled if: true
    Ellipse (460,333 34x34), colour toggle: PR_Line01.fb_Transfer.fbCylinder_Comb.bAtRetract, input disabled if: true
    Ellipse (460,388 34x34), colour toggle: PR_Line01.fb_Transfer.fbCylinder_Comb.bAtExtend, input disabled if: true
    Ellipse (460,443 34x34), colour toggle: PR_Line01.fb_Transfer.fbCylinder_Move_Comb.bAtRetract, input disabled if: true
    Ellipse (460,498 34x34), colour toggle: PR_Line01.fb_Transfer.fbCylinder_Move_Comb.bAtExtend, input disabled if: true
    Rectangle (513,215 450x50), "U1I7-5. Cảm biến đẩy ra của ben kẹp hũ"
    Rectangle (513,160 450x50), "U1I7-4. Cảm biến rút về của ben kẹp hũ"
    Rectangle (513,270 450x50), "U1I7-6. Cảm biến phát hiện hũ ở chỗ cân thức ăn"
    Rectangle (513,325 450x50), "U1I7-7. Cảm biến phát hiện hũ ở chỗ cân sâu"
    Rectangle (513,380 450x50), "U1I7-8. Cảm biến cửa 1"
    Rectangle (513,435 450x50), "U1I7-9. Cảm biến cửa 2"
    Rectangle (513,490 450x50), "U1I7-10. Cảm biến cửa 3"
    Ellipse (975,168 34x34), colour toggle: PR_Line01.fb_Transfer.fbCylinder_Clip.bAtExtend, input disabled if: true
    Ellipse (975,223 34x34), colour toggle: PR_Line01.fb_Transfer.fbCylinder_Clip.bAtRetract, input disabled if: true
    Ellipse (975,278 34x34), colour toggle: PR_Line01.fb_FoodWeight.bCupPresent, input disabled if: true
    Ellipse (975,333 34x34), colour toggle: PR_Line01.fb_WormWeight.bCupPresent, input disabled if: true
    Ellipse (975,388 34x34), colour toggle: GVL_IO.bSafetyDoor1, input disabled if: true
    Ellipse (975,443 34x34), colour toggle: GVL_IO.bSafetyDoor2, input disabled if: true
    Ellipse (975,498 34x34), colour toggle: GVL_IO.bSafetyDoor3, input disabled if: true
    Image (953,101 70x50), image: ImagePool.Qua trai
        OnMouseClick: change screen: N_PLC_I1
    Rectangle (0,61 341x40), "INPUT"
        OnMouseClick: change screen: N_PLC_I1
    Rectangle (341,61 341x40), "OUTPUT"
        OnMouseClick: change screen: N_PLC_O1
    Rectangle (682,61 341x40), "PARAMETER"
        OnMouseClick: change screen: N_Parameter_1
END_VISUALIZATION

// ---- VISUs/IO/N_PLC_I2.TcVIS
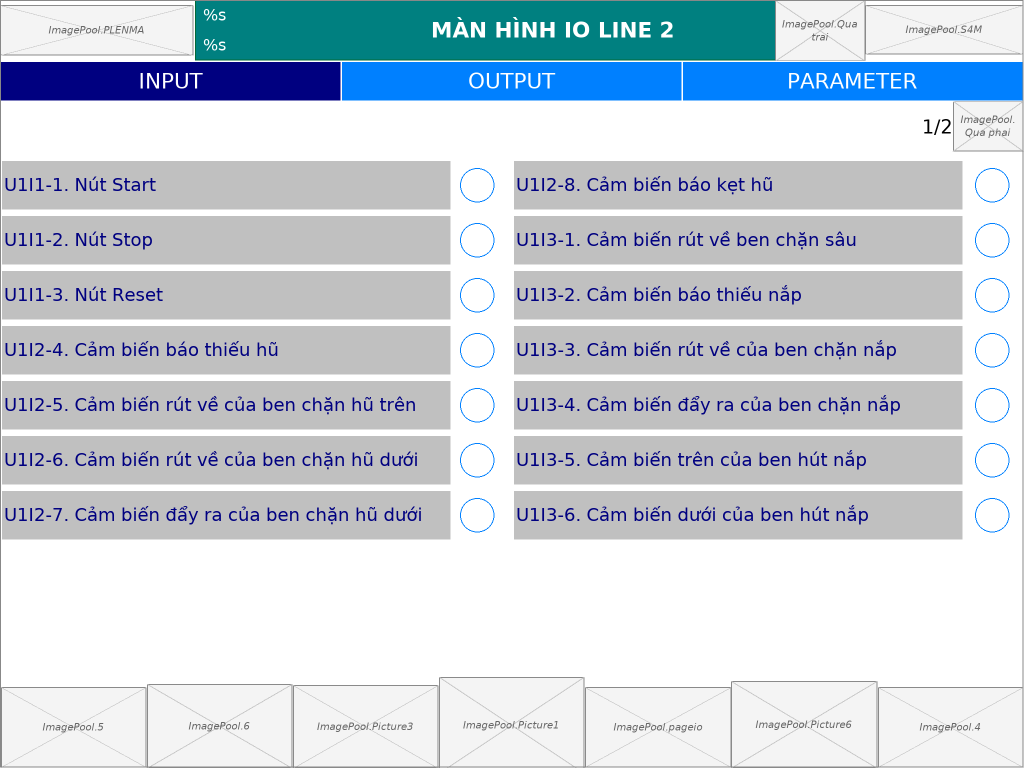
VISUALIZATION N_PLC_I2  // 1024x768
    Rectangle (886,102 103x50), "1/2"
    Frame (0,687 1024x80)
        shows N_Footer_Line2()
    Frame (0,0 1024x60)
        shows N_Header()
    Textfield (353,5 400x50), "MÀN HÌNH IO LINE 2"
    Image (775,0 90x61), image: ImagePool.Qua trai
        OnMouseClick: change screen: N_PLC_I1
    Rectangle (1,325 450x50), "U1I2-4. Cảm biến báo thiếu hũ"
    Rectangle (1,380 450x50), "U1I2-5. Cảm biến rút về của ben chặn hũ trên"
    Rectangle (1,435 450x50), "U1I2-6. Cảm biến rút về của ben chặn hũ dưới"
    Rectangle (1,490 450x50), "U1I2-7. Cảm biến đẩy ra của ben chặn hũ dưới"
    Rectangle (1,160 450x50), "U1I1-1. Nút Start"
    Rectangle (1,215 450x50), "U1I1-2. Nút Stop"
    Rectangle (1,270 450x50), "U1I1-3. Nút Reset"
    Ellipse (460,168 34x34), colour toggle: GVL_IO.bStart, input disabled if: true
    Ellipse (460,223 34x34), colour toggle: GVL_IO.bStop, input disabled if: true
    Ellipse (460,278 34x34), colour toggle: GVL_IO.bReset, input disabled if: true
    Ellipse (460,333 34x34), colour toggle: PR_Line02.fb_CupSupply.bCupEmpty, input disabled if: true
    Ellipse (460,388 34x34), colour toggle: PR_Line02.fb_CupSupply.fbCylinder_Up.bAtRetract, input disabled if: true
    Ellipse (460,443 34x34), colour toggle: PR_Line02.fb_CupSupply.fbCylinder_Dw.bAtRetract, input disabled if: true
    Ellipse (460,498 34x34), colour toggle: PR_Line02.fb_CupSupply.fbCylinder_Dw.bAtExtend, input disabled if: true
    Rectangle (513,490 450x50), "U1I3-6. Cảm biến dưới của ben hút nắp"
    Rectangle (513,160 450x50), "U1I2-8. Cảm biến báo kẹt hũ"
    Rectangle (513,215 450x50), "U1I3-1. Cảm biến rút về ben chặn sâu"
    Rectangle (513,270 450x50), "U1I3-2. Cảm biến báo thiếu nắp"
    Rectangle (513,325 450x50), "U1I3-3. Cảm biến rút về của ben chặn nắp"
    Rectangle (513,380 450x50), "U1I3-4. Cảm biến đẩy ra của ben chặn nắp"
    Rectangle (513,435 450x50), "U1I3-5. Cảm biến trên của ben hút nắp"
    Ellipse (975,168 34x34), colour toggle: PR_Line02.fb_CupSupply.bCupDrop, input disabled if: true
    Ellipse (975,498 34x34), colour toggle: PR_Line02.fb_LidSupply.fbCylinder_Suction.bAtExtend, input disabled if: true
    Ellipse (975,223 34x34), colour toggle: PR_Line02.fb_WormWeight.fbCylinder.bAtRetract, input disabled if: true
    Ellipse (975,278 34x34), colour toggle: PR_Line02.fb_LidSupply.bLidEmpty, input disabled if: true
    Ellipse (975,333 34x34), colour toggle: PR_Line02.fb_LidSupply.fbCylinder_LidStopper.bAtRetract, input disabled if: true
    Ellipse (975,388 34x34), colour toggle: PR_Line02.fb_LidSupply.fbCylinder_LidStopper.bAtExtend, input disabled if: true
    Ellipse (975,443 34x34), colour toggle: PR_Line02.fb_LidSupply.fbCylinder_Suction.bAtRetract, input disabled if: true
    Image (953,101 70x50), image: ImagePool.Qua phai
        OnMouseClick: change screen: N_PLC_I2_next
    Rectangle (0,61 341x40), "INPUT"
        OnMouseClick: change screen: N_PLC_I2
    Rectangle (341,61 341x40), "OUTPUT"
        OnMouseClick: change screen: N_PLC_O2
    Rectangle (682,61 341x40), "PARAMETER"
        OnMouseClick: change screen: N_Parameter_2
END_VISUALIZATION

// ---- VISUs/IO/N_PLC_I2_next.TcVIS
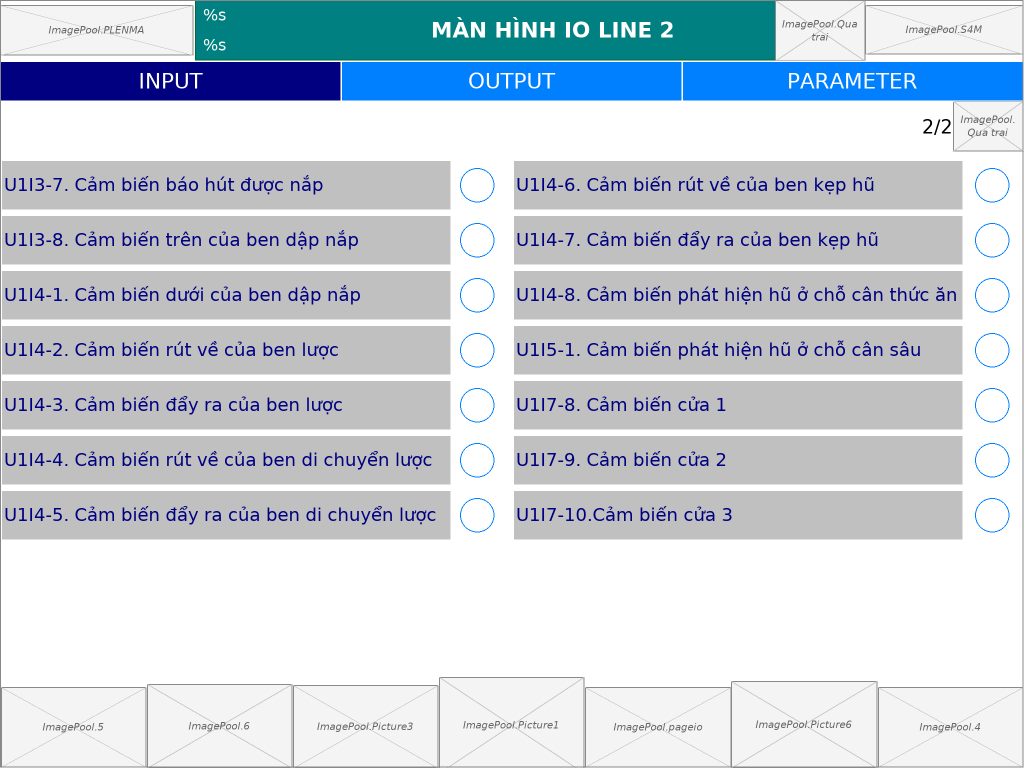
VISUALIZATION N_PLC_I2_next  // 1024x768
    Rectangle (886,102 103x50), "2/2"
    Frame (0,687 1024x80)
        shows N_Footer_Line2()
    Frame (0,0 1024x60)
        shows N_Header()
    Textfield (353,5 400x50), "MÀN HÌNH IO LINE 2"
    Image (775,0 90x61), image: ImagePool.Qua trai
        OnMouseClick: change screen: N_PLC_I2
    Rectangle (1,160 450x50), "U1I3-7. Cảm biến báo hút được nắp"
    Rectangle (1,215 450x50), "U1I3-8. Cảm biến trên của ben dập nắp"
    Rectangle (1,325 450x50), "U1I4-2. Cảm biến rút về của ben lược"
    Rectangle (1,270 450x50), "U1I4-1. Cảm biến dưới của ben dập nắp"
    Rectangle (1,380 450x50), "U1I4-3. Cảm biến đẩy ra của ben lược"
    Rectangle (1,435 450x50), "U1I4-4. Cảm biến rút về của ben di chuyển lược"
    Rectangle (1,490 450x50), "U1I4-5. Cảm biến đẩy ra của ben di chuyển lược"
    Ellipse (460,168 34x34), colour toggle: PR_Line02.fb_LidSupply.fbLidSuctionValve.bPressure, input disabled if: true
    Ellipse (460,223 34x34), colour toggle: PR_Line02.fb_LidClose.fbCylinder_LidClose.bAtRetract, input disabled if: true
    Ellipse (460,278 34x34), colour toggle: PR_Line02.fb_LidClose.fbCylinder_LidClose.bAtExtend, input disabled if: true
    Ellipse (460,333 34x34), colour toggle: PR_Line02.fb_Transfer.fbCylinder_Comb.bAtRetract, input disabled if: true
    Ellipse (460,388 34x34), colour toggle: PR_Line02.fb_Transfer.fbCylinder_Comb.bAtExtend, input disabled if: true
    Ellipse (460,443 34x34), colour toggle: PR_Line02.fb_Transfer.fbCylinder_Move_Comb.bAtRetract, input disabled if: true
    Ellipse (460,498 34x34), colour toggle: PR_Line02.fb_Transfer.fbCylinder_Move_Comb.bAtExtend, input disabled if: true
    Rectangle (513,215 450x50), "U1I4-7. Cảm biến đẩy ra của ben kẹp hũ"
    Rectangle (513,160 450x50), "U1I4-6. Cảm biến rút về của ben kẹp hũ"
    Rectangle (513,270 450x50), "U1I4-8. Cảm biến phát hiện hũ ở chỗ cân thức ăn"
    Rectangle (513,325 450x50), "U1I5-1. Cảm biến phát hiện hũ ở chỗ cân sâu"
    Rectangle (513,380 450x50), "U1I7-8. Cảm biến cửa 1"
    Rectangle (513,435 450x50), "U1I7-9. Cảm biến cửa 2"
    Rectangle (513,490 450x50), "U1I7-10.Cảm biến cửa 3"
    Ellipse (975,168 34x34), colour toggle: PR_Line02.fb_Transfer.fbCylinder_Clip.bAtRetract, input disabled if: true
    Ellipse (975,223 34x34), colour toggle: PR_Line02.fb_Transfer.fbCylinder_Clip.bAtRetract, input disabled if: true
    Ellipse (975,278 34x34), colour toggle: PR_Line02.fb_FoodWeight.bCupPresent, input disabled if: true
    Ellipse (975,333 34x34), colour toggle: PR_Line02.fb_WormWeight.bCupPresent, input disabled if: true
    Ellipse (975,388 34x34), colour toggle: GVL_IO.bSafetyDoor1, input disabled if: true
    Ellipse (975,443 34x34), colour toggle: GVL_IO.bSafetyDoor2, input disabled if: true
    Ellipse (975,498 34x34), colour toggle: GVL_IO.bSafetyDoor3, input disabled if: true
    Image (953,101 70x50), image: ImagePool.Qua trai
        OnMouseClick: change screen: N_PLC_I2
    Rectangle (0,61 341x40), "INPUT"
        OnMouseClick: change screen: N_PLC_I2
    Rectangle (341,61 341x40), "OUTPUT"
        OnMouseClick: change screen: N_PLC_O2
    Rectangle (682,61 341x40), "PARAMETER"
        OnMouseClick: change screen: N_Parameter_2
END_VISUALIZATION

// ---- VISUs/IO/N_PLC_O1.TcVIS
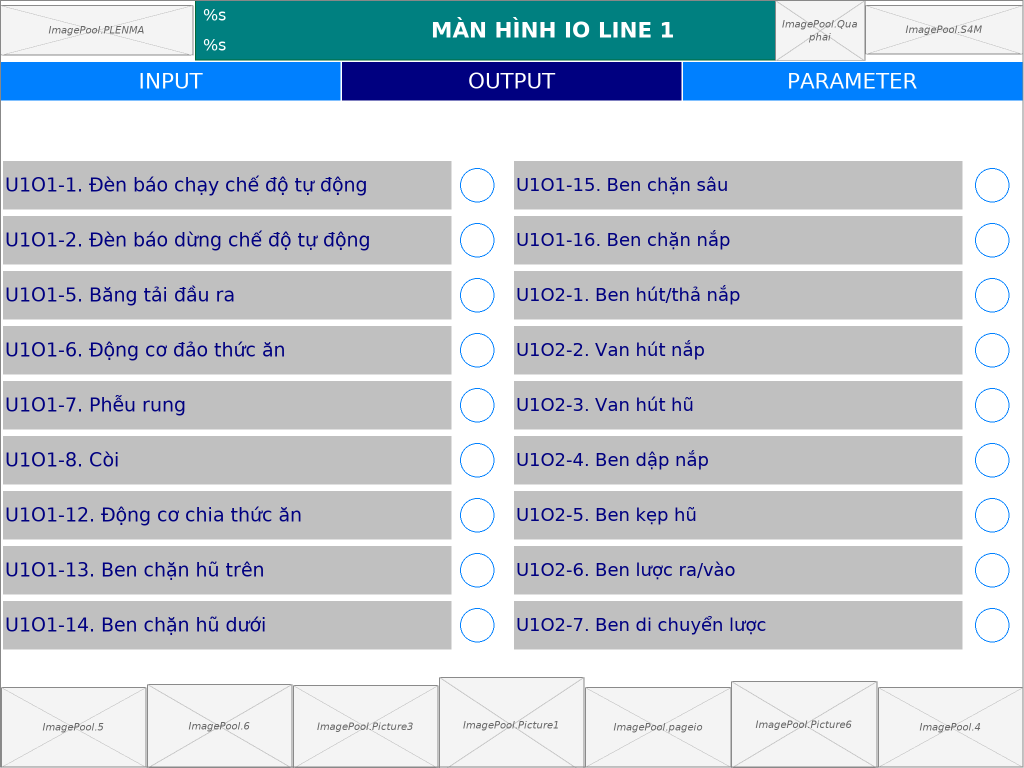
VISUALIZATION N_PLC_O1  // 1024x768
    Frame (0,687 1024x80)
        shows N_Footer_Line1()
    Frame (0,0 1024x60)
        shows N_Header()
    Textfield (353,5 400x50), "MÀN HÌNH IO LINE 1"
    Image (775,0 90x61), image: ImagePool.Qua phai
        OnMouseClick: change screen: N_PLC_O2
    Rectangle (2,160 450x50), "U1O1-1. Đèn báo chạy chế độ tự động"
    Rectangle (2,215 450x50), "U1O1-2. Đèn báo dừng chế độ tự động"
    Rectangle (2,270 450x50), "U1O1-5. Băng tải đầu ra"
    Ellipse (460,168 34x34), colour toggle: GVL_IO.bLight_Running, input disabled if: true
    Ellipse (460,223 34x34), colour toggle: GVL_IO.bLight_Stop, input disabled if: true
    Rectangle (2,325 450x50), "U1O1-6. Động cơ đảo thức ăn"
    Rectangle (2,380 450x50), "U1O1-7. Phễu rung"
    Rectangle (2,435 450x50), "U1O1-8. Còi"
    Rectangle (2,490 450x50), "U1O1-12. Động cơ chia thức ăn"
    Rectangle (2,545 450x50), "U1O1-13. Ben chặn hũ trên"
    Rectangle (2,600 450x50), "U1O1-14. Ben chặn hũ dưới"
    Rectangle (513,160 450x50), "U1O1-15. Ben chặn sâu"
    Rectangle (513,215 450x50), "U1O1-16. Ben chặn nắp"
    Ellipse (460,278 34x34), colour toggle: PR_Conveyor_Out.fb_Conveyor.fbInverter.bVFD, input disabled if: true
    Ellipse (460,333 34x34), colour toggle: PR_Line01.fb_FoodMixer.fbInverter.bVFD, input disabled if: true
    Ellipse (460,388 34x34), colour toggle: PR_Line01.fb_WormWeight.fbInverter.bVFD, input disabled if: true
    Ellipse (460,443 34x34), colour toggle: GVL_IO.bSirens, input disabled if: true
    Ellipse (460,498 34x34), colour toggle: PR_Line01.fb_FoodWeight.fbDriver.bVFD, input disabled if: true
    Ellipse (460,553 34x34), colour toggle: PR_Line01.fb_CupSupply.fbCylinder_Up.bMoveExtend, input disabled if: true
    Ellipse (460,608 34x34), colour toggle: PR_Line01.fb_CupSupply.fbCylinder_Dw.bMoveRetract, input disabled if: true
    Ellipse (975,168 34x34), colour toggle: PR_Line02.fb_WormWeight.fbCylinder.bMoveRetract, input disabled if: true
    Ellipse (975,223 34x34), colour toggle: PR_Line01.fb_LidSupply.fbCylinder_LidStopper.bMoveRetract, input disabled if: true
    Rectangle (513,270 450x50), "U1O2-1. Ben hút/thả nắp"
    Ellipse (975,278 34x34), colour toggle: PR_Line02.fb_LidSupply.fbCylinder_Suction.bMoveExtend, input disabled if: true
    Rectangle (513,325 450x50), "U1O2-2. Van hút nắp"
    Rectangle (513,380 450x50), "U1O2-3. Van hút hũ"
    Rectangle (513,435 450x50), "U1O2-4. Ben dập nắp"
    Rectangle (513,490 450x50), "U1O2-5. Ben kẹp hũ"
    Rectangle (513,545 450x50), "U1O2-6. Ben lược ra/vào"
    Rectangle (513,600 450x50), "U1O2-7. Ben di chuyển lược"
    Ellipse (975,333 34x34), colour toggle: PR_Line02.fb_LidSupply.fbLidSuctionValve.bSuck, input disabled if: true
    Ellipse (975,388 34x34), colour toggle: PR_Line02.fb_LidSupply.fbCupSuctionValve.bSuck, input disabled if: true
    Ellipse (975,443 34x34), colour toggle: PR_Line02.fb_LidClose.fbCylinder_LidClose.bMoveExtend, input disabled if: true
    Ellipse (975,498 34x34), colour toggle: PR_Line01.fb_Transfer.fbCylinder_Clip.bMoveRetract, input disabled if: true
    Ellipse (975,553 34x34), colour toggle: PR_Line01.fb_Transfer.fbCylinder_Comb.bMoveExtend, input disabled if: true
    Ellipse (975,608 34x34), colour toggle: PR_Line01.fb_Transfer.fbCylinder_Move_Comb.bMoveExtend, input disabled if: true
    Rectangle (0,61 341x40), "INPUT"
        OnMouseClick: change screen: N_PLC_I1
    Rectangle (341,61 341x40), "OUTPUT"
        OnMouseClick: change screen: N_PLC_O1
    Rectangle (682,61 341x40), "PARAMETER"
        OnMouseClick: change screen: N_Parameter_1
END_VISUALIZATION

// ---- VISUs/IO/N_PLC_O2.TcVIS
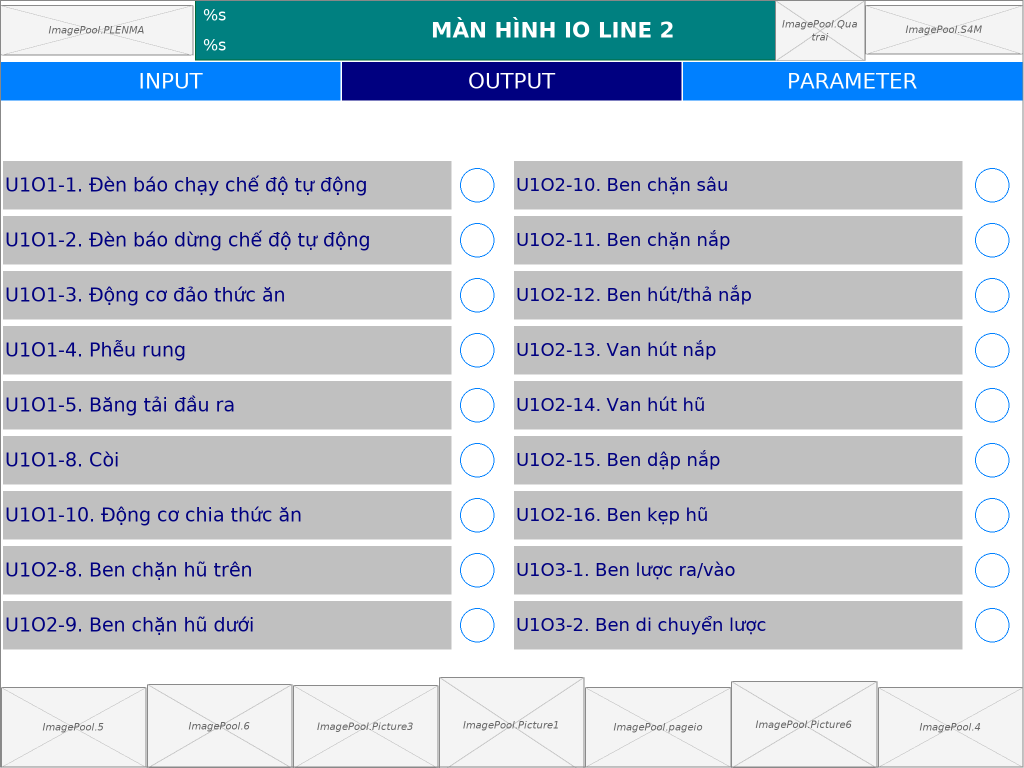
VISUALIZATION N_PLC_O2  // 1024x768
    Frame (0,687 1024x80)
        shows N_Footer_Line2()
    Frame (0,0 1024x60)
        shows N_Header()
    Textfield (353,5 400x50), "MÀN HÌNH IO LINE 2"
    Rectangle (2,160 450x50), "U1O1-1. Đèn báo chạy chế độ tự động"
    Rectangle (2,215 450x50), "U1O1-2. Đèn báo dừng chế độ tự động"
    Rectangle (2,270 450x50), "U1O1-3. Động cơ đảo thức ăn"
    Ellipse (460,168 34x34), colour toggle: GVL_IO.bLight_Running, input disabled if: true
    Ellipse (460,223 34x34), colour toggle: GVL_IO.bLight_Stop, input disabled if: true
    Rectangle (2,325 450x50), "U1O1-4. Phễu rung"
    Rectangle (2,380 450x50), "U1O1-5. Băng tải đầu ra"
    Rectangle (2,435 450x50), "U1O1-8. Còi"
    Rectangle (2,490 450x50), "U1O1-10. Động cơ chia thức ăn"
    Rectangle (2,545 450x50), "U1O2-8. Ben chặn hũ trên"
    Rectangle (2,600 450x50), "U1O2-9. Ben chặn hũ dưới"
    Rectangle (513,160 450x50), "U1O2-10. Ben chặn sâu"
    Rectangle (513,215 450x50), "U1O2-11. Ben chặn nắp"
    Ellipse (460,278 34x34), colour toggle: PR_Line02.fb_FoodMixer.fbInverter.bVFD, input disabled if: true
    Ellipse (460,333 34x34), colour toggle: PR_Line02.fb_WormWeight.fbInverter.bVFD, input disabled if: true
    Ellipse (460,388 34x34), colour toggle: PR_Conveyor_Out.fb_Conveyor.fbInverter.bVFD, input disabled if: true
    Ellipse (460,443 34x34), colour toggle: GVL_IO.bSirens, input disabled if: true
    Ellipse (460,498 34x34), input disabled if: true
    Ellipse (460,553 34x34), colour toggle: PR_Line02.fb_CupSupply.fbCylinder_Up.bMoveExtend, input disabled if: true
    Ellipse (460,608 34x34), colour toggle: PR_Line02.fb_CupSupply.fbCylinder_Dw.bMoveRetract, input disabled if: true
    Ellipse (975,168 34x34), input disabled if: true
    Ellipse (975,223 34x34), colour toggle: PR_Line02.fb_LidSupply.fbCylinder_LidStopper.bMoveRetract, input disabled if: true
    Rectangle (513,270 450x50), "U1O2-12. Ben hút/thả nắp"
    Ellipse (975,278 34x34), input disabled if: true
    Rectangle (513,325 450x50), "U1O2-13. Van hút nắp"
    Rectangle (513,380 450x50), "U1O2-14. Van hút hũ"
    Rectangle (513,435 450x50), "U1O2-15. Ben dập nắp"
    Rectangle (513,490 450x50), "U1O2-16. Ben kẹp hũ"
    Rectangle (513,545 450x50), "U1O3-1. Ben lược ra/vào"
    Rectangle (513,600 450x50), "U1O3-2. Ben di chuyển lược"
    Ellipse (975,333 34x34), input disabled if: true
    Ellipse (975,388 34x34), input disabled if: true
    Ellipse (975,443 34x34), input disabled if: true
    Ellipse (975,498 34x34), colour toggle: PR_Line02.fb_Transfer.fbCylinder_Clip.bMoveRetract, input disabled if: true
    Ellipse (975,553 34x34), colour toggle: PR_Line02.fb_Transfer.fbCylinder_Comb.bMoveExtend, input disabled if: true
    Ellipse (975,608 34x34), colour toggle: PR_Line02.fb_Transfer.fbCylinder_Move_Comb.bMoveExtend, input disabled if: true
    Image (775,0 90x61), image: ImagePool.Qua trai
        OnMouseClick: change screen: N_PLC_O1
    Rectangle (0,61 341x40), "INPUT"
        OnMouseClick: change screen: N_PLC_I2
    Rectangle (341,61 341x40), "OUTPUT"
        OnMouseClick: change screen: N_PLC_O2
    Rectangle (682,61 341x40), "PARAMETER"
        OnMouseClick: change screen: N_Parameter_2
END_VISUALIZATION

// ---- VISUs/Main_Line/MAIN_LINE1.TcVIS
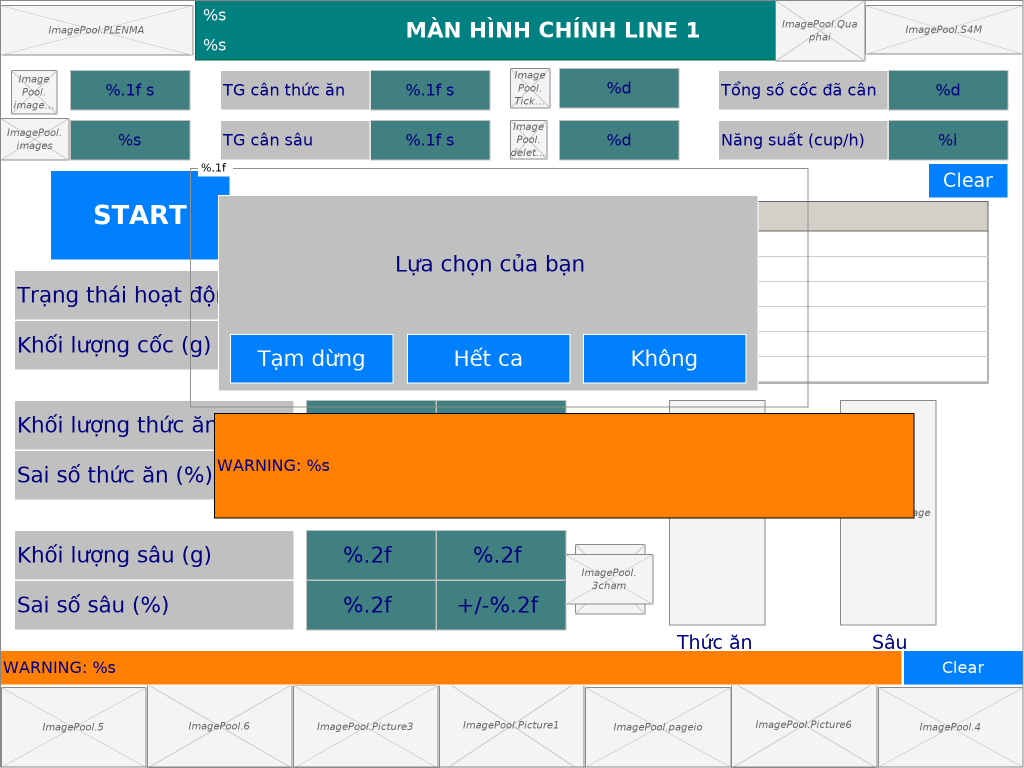
VISUALIZATION MAIN_LINE1  // 1024x768
    Rectangle (50,170 180x90), "STOP", invisible if: not bStatusStart1, input disabled if: not bStatusStart1
        OnMouseDown: execute { hienthiDialog := TRUE; }
    Rectangle (50,170 180x90), "START", invisible if: bStatusStart1, input disabled if: Not brunauto
        OnMouseDown: execute { bStart1 := true; }
    Table (615,201 373x182), data array: PR_Line01.fProductLog
        p3854506369: PR_Line01.fProductLog[1][INDEX]
        p1892666644: PR_Line01.fProductLog[2][INDEX]
        p2232123230: Thức ăn
        p511219082: Sâu
    RoundedRectangle (840,625 100x35), "Sâu"
    RoundedRectangle (665,625 100x35), "Thức ăn"
    Rectangle (306,400 130x50), "%.2f", text variable: PR_Line01.fb_FoodWeight.fWeight_Food
    Rectangle (306,450 130x50), "%.2f", text variable: PR_Line01.fb_FoodWeight.fActDelta_Food
    Rectangle (306,320 260x50), "%.2f", text variable: PR_Line01.fb_FoodWeight.fTareWeight
    Rectangle (436,400 130x50), "%.2f", text variable: PR_Line01.fDerisedWeight_Food
    Rectangle (436,450 130x50), "+/-%.2f", text variable: PR_Line01.fDelta_Food
    Rectangle (306,200 130x60), "Thực tế"
    Rectangle (306,270 260x50), "%s", text variable: nStatus1
    Rectangle (437,200 130x60), "Cài đặt"
    Rectangle (306,530 130x50), "%.2f", text variable: PR_Line01.fb_WormWeight.fWeight_Worm
    Rectangle (306,580 130x50), "%.2f", text variable: PR_Line01.fb_WormWeight.fActDelta_Worm
    Rectangle (436,530 130x50), "%.2f", text variable: PR_Line01.fDerisedWeight_Worm
    Rectangle (436,580 130x50), "+/-%.2f", text variable: PR_Line01.fDelta_Worm
    BarDisplayImage (669,400 96x225), value: PR_Line01.fb_FoodWeight.fWeight_Food, style: BarDisplayImage-Gray, scale format: %.1f, scale 0..18
    BarDisplayImage (840,400 96x225), value: PR_Line01.fb_WormWeight.fWeight_Worm, style: BarDisplayImage-Gray, scale format: %.1f, scale 0..5
    Frame (0,687 1024x80)
        shows N_Footer_Line1()
    Frame (0,0 1024x60)
        shows N_Header()
    Rectangle (14,270 280x50), "Trạng thái hoạt động"
    Rectangle (14,530 280x50), "Khối lượng sâu (g)"
    Rectangle (14,580 280x50), "Sai số sâu (%)"
    Rectangle (14,320 280x50), "Khối lượng cốc (g)"
    Rectangle (14,450 280x50), "Sai số thức ăn (%)"
    Rectangle (14,400 280x50), "Khối lượng thức ăn (g)"
    Textfield (353,5 400x50), "MÀN HÌNH CHÍNH LINE 1"
    Image (775,0 90x61), image: ImagePool.Qua phai
        OnMouseClick: change screen: MAIN_LINE2
        OnMouseClick: execute { MAIN_LINE2.bModeAuto := TRUE; MAIN_LINE2.bModeManual := FALSE; }
    ImageSwitcher (575,414 70x70), variable: PR_Line01.fb_FoodWeight.bStatus_Food, invisible if: not PR_Line01.fb_FoodWeight.bStatus, input disabled if: true, background image: ImagePool.262-2627516_clipart-cross-tick-green-tick-png-icon, image: ImagePool.delete-button-png-28575, behaviour: TOGGLE
    ImageSwitcher (575,544 70x70), variable: PR_Line01.fb_WormWeight.bStatus_Worm, invisible if: not PR_Line01.fb_WormWeight.bStatus, input disabled if: true, background image: ImagePool.262-2627516_clipart-cross-tick-green-tick-png-icon, image: ImagePool.delete-button-png-28575, behaviour: TOGGLE
    Frame (0,650 1024x35)
        shows N_Footer_Alarm()
    Rectangle (70,70 120x40), "%.1f s", text variable: PR_Line01.timeCycle
    Rectangle (370,70 120x40), "%.1f s", text variable: PR_Line01.fb_FoodWeight.fTime
    Image (11,70 46x44), image: ImagePool.images (1)
    Rectangle (70,120 120x40), "%s", text variable: PRG_MainRecipe1.RecipeName
    Image (0,118 69x42), image: ImagePool.images
    Rectangle (888,70 120x40), "%d", text variable: nCount1
    Image (510,68 40x40), image: ImagePool.Tick-Green-Check-Mark-PNG-Clipart
    Rectangle (559,68 120x40), "%d", text variable: nResult_true1
    Image (510,120 37x39), image: ImagePool.delete-button-png-28575
    Rectangle (559,120 120x40), "%d", text variable: nResult_false1
    Rectangle (928,163 80x35), "Clear"
        tap GVL_OF_VU.bClear[2]
        OnMouseDown: execute { bClear1 := true; }
    Rectangle (370,120 120x40), "%.1f s", text variable: PR_Line01.fb_WormWeight.fTime
    Rectangle (888,120 120x40), "%i", text variable: PR_Line01.fproduct
    Rectangle (718,70 170x40), "Tổng số cốc đã cân"
    Rectangle (220,70 150x40), "TG cân thức ăn"
    Rectangle (220,120 150x40), "TG cân sâu"
    Rectangle (718,120 170x40), "Năng suất (cup/h)"
    Image (565,554 88x50), invisible if: PR_Line01.fb_WormWeight.bStatus, image: ImagePool.3cham
    Image (565,423 88x50), invisible if: PR_Line01.fb_FoodWeight.bStatus, image: ImagePool.3cham
    GroupBox (190,160 618x247), "%.1f", invisible if: not hienthiDialog, input disabled if: not hienthiDialog
        Rectangle (28,35 540x196), invisible if: not hienthiDialog, input disabled if: not hienthiDialog
        Rectangle (393,174 163x49), "Không", invisible if: not hienthiDialog, input disabled if: not hienthiDialog
            OnMouseDown: execute { hienthiDialog := FALSE; }
        Label (107,78 386x52), "Lựa chọn của bạn", invisible if: not hienthiDialog
        Rectangle (40,174 163x49), "Tạm dừng", input disabled if: not hienthiDialog
            OnMouseDown: execute { bStop1 := TRUE; hienthiDialog := FALSE; }
        Rectangle (217,174 163x49), "Hết ca", invisible if: not hienthiDialog, input disabled if: not hienthiDialog
            OnMouseDown: execute { bShift_is_over1 := TRUE; hienthiDialog := FALSE; }
    Rectangle (214,413 700x105), "WARNING: %s", text variable: stWarningTxt2, invisible if: not bAlarm_Iot, input disabled if: not bAlarm_Iot
END_VISUALIZATION

// ---- VISUs/Main_Line/MAIN_LINE2.TcVIS
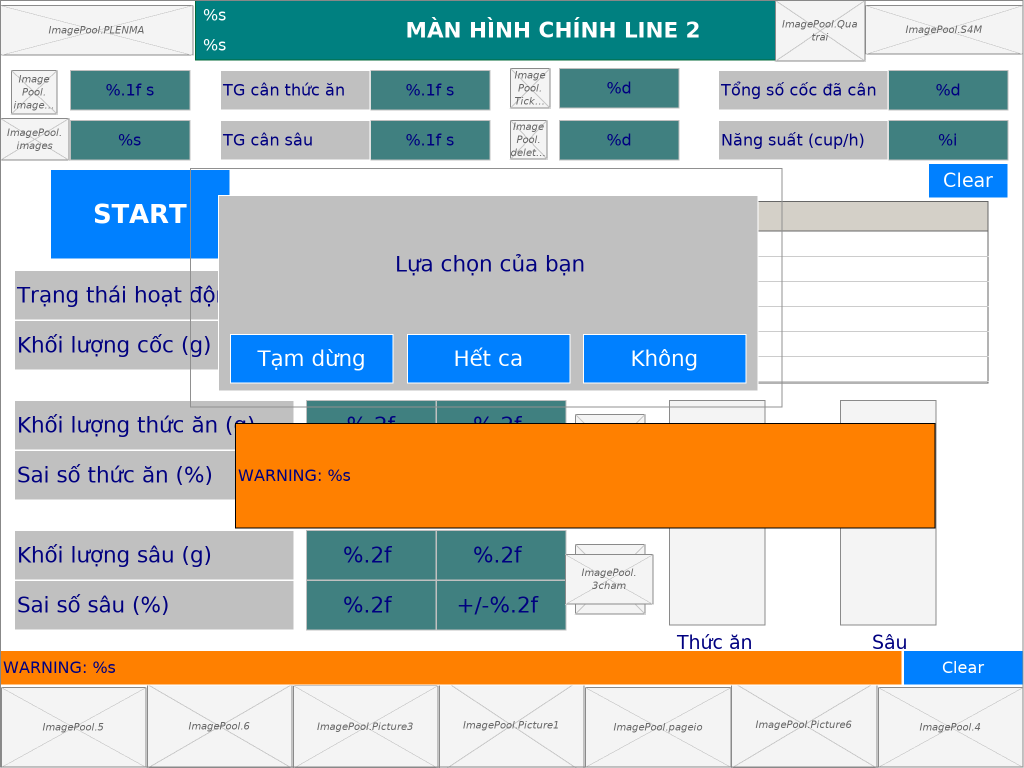
VISUALIZATION MAIN_LINE2  // 1024x768
    Rectangle (49,168 180x90), "STOP", invisible if: not bStatusStart2, input disabled if: not bStatusStart2
        OnMouseDown: execute { hienthiDialog2 := TRUE; }
    Rectangle (50,169 180x90), "START", invisible if: bStatusStart2, input disabled if: Not bRunAuto
        OnMouseDown: execute { bStart2 := true; }
    Frame (0,687 1024x80)
        shows N_Footer_Line2()
    Frame (0,0 1024x60)
        shows N_Header()
    Textfield (353,5 400x50), "MÀN HÌNH CHÍNH LINE 2"
    Rectangle (70,70 120x40), "%.1f s", text variable: PR_Line02.timeCycle
    Rectangle (370,70 120x40), "%.1f s", text variable: PR_Line02.fb_FoodWeight.fTime
    Image (11,70 46x44), image: ImagePool.images (1)
    Rectangle (70,120 120x40), "%s", text variable: PRG_MainRecipe1_1.RecipeName
    Image (0,118 69x42), image: ImagePool.images
    Rectangle (888,70 120x40), "%d", text variable: nCount2
    Image (510,68 40x40), image: ImagePool.Tick-Green-Check-Mark-PNG-Clipart
    Rectangle (559,68 120x40), "%d", text variable: nResult_true2
    Image (510,120 37x39), image: ImagePool.delete-button-png-28575
    Rectangle (559,120 120x40), "%d", text variable: nResult_false2
    Rectangle (928,163 80x35), "Clear"
        tap GVL_OF_VU.bClear[2]
        OnMouseDown: execute { bClear2 := true; }
    Rectangle (370,120 120x40), "%.1f s", text variable: PR_Line02.fb_WormWeight.fTime
    Image (775,0 90x61), image: ImagePool.Qua trai
        OnMouseClick: change screen: MAIN_LINE1
        OnMouseClick: execute { MAIN.bModeAuto := TRUE; MAIN.bModeManual := FALSE; }
    RoundedRectangle (840,625 100x35), "Sâu"
    RoundedRectangle (665,625 100x35), "Thức ăn"
    Rectangle (306,400 130x50), "%.2f", text variable: PR_Line02.fb_FoodWeight.fWeight_Food
    Rectangle (306,450 130x50), "%.2f", text variable: PR_Line02.fb_FoodWeight.fActDelta_Food
    Rectangle (306,320 260x50), "%.2f", text variable: PR_Line02.fb_FoodWeight.fTareWeight
    Rectangle (436,400 130x50), "%.2f", text variable: PR_Line02.fDerisedWeight_Food
    Rectangle (436,450 130x50), "+/-%.2f", text variable: PR_Line02.fDelta_Food
    Rectangle (306,200 130x60), "Thực tế"
    Rectangle (306,270 260x50), "%s", text variable: nStatus2
    Rectangle (437,200 130x60), "Cài đặt"
    Rectangle (306,530 130x50), "%.2f", text variable: PR_Line02.fb_WormWeight.fWeight_Worm
    Rectangle (306,580 130x50), "%.2f", text variable: PR_Line02.fb_WormWeight.fActDelta_Worm
    Rectangle (436,530 130x50), "%.2f", text variable: PR_Line02.fDerisedWeight_Worm
    Rectangle (436,580 130x50), "+/-%.2f", text variable: PR_Line02.fDelta_Worm
    BarDisplayImage (669,400 96x225), value: PR_Line02.fb_FoodWeight.fWeight_Food, style: BarDisplayImage-Gray, scale format: %.1f, scale 0..18
    BarDisplayImage (840,400 96x225), value: PR_Line02.fb_WormWeight.fWeight_Worm, style: BarDisplayImage-Gray, scale format: %.1f, scale 0..5
    Rectangle (14,270 280x50), "Trạng thái hoạt động"
    Rectangle (14,530 280x50), "Khối lượng sâu (g)"
    Rectangle (14,580 280x50), "Sai số sâu (%)"
    Rectangle (14,320 280x50), "Khối lượng cốc (g)"
    Rectangle (14,450 280x50), "Sai số thức ăn (%)"
    Rectangle (14,400 280x50), "Khối lượng thức ăn (g)"
    ImageSwitcher (575,414 70x70), variable: PR_Line02.fb_FoodWeight.bStatus_Food, invisible if: not PR_Line02.fb_FoodWeight.bStatus, input disabled if: true, background image: ImagePool.262-2627516_clipart-cross-tick-green-tick-png-icon, image: ImagePool.delete-button-png-28575, behaviour: TOGGLE
    ImageSwitcher (575,544 70x70), variable: PR_Line02.fb_WormWeight.bStatus_Worm, invisible if: not PR_Line02.fb_WormWeight.bStatus, input disabled if: true, background image: ImagePool.262-2627516_clipart-cross-tick-green-tick-png-icon, image: ImagePool.delete-button-png-28575, behaviour: TOGGLE
    Table (615,201 373x182), data array: PR_Line02.fProductLog
        p3854506369: PR_Line02.fProductLog[1][INDEX]
        p1892666644: PR_Line02.fProductLog[2][INDEX]
        p2232123230: Thức ăn
        p511219082: Sâu
    Frame (0,650 1024x35)
        shows N_Footer_Alarm_1()
    Rectangle (888,120 120x40), "%i", text variable: PR_Line02.fproduct
    Rectangle (718,70 170x40), "Tổng số cốc đã cân"
    Rectangle (220,70 150x40), "TG cân thức ăn"
    Rectangle (220,120 150x40), "TG cân sâu"
    Rectangle (718,120 170x40), "Năng suất (cup/h)"
    Image (565,554 88x50), invisible if: PR_Line02.fb_WormWeight.bStatus, image: ImagePool.3cham
    Image (565,424 88x50), invisible if: PR_Line02.fb_FoodWeight.bStatus, image: ImagePool.3cham
    GroupBox (190,160 592x247), invisible if: not hienthiDialog2, input disabled if: not hienthiDialog2
        Rectangle (28,35 540x196), invisible if: not hienthiDialog2, input disabled if: not hienthiDialog2
        Rectangle (393,174 163x49), "Không", invisible if: not hienthiDialog2, input disabled if: not hienthiDialog2
            OnMouseDown: execute { hienthiDialog2 := FALSE; }
        Label (107,78 386x52), "Lựa chọn của bạn", invisible if: not hienthiDialog
        Rectangle (40,174 163x49), "Tạm dừng", input disabled if: not hienthiDialog2
            OnMouseDown: execute { bStop2 := TRUE; hienthiDialog2 := FALSE; }
        Rectangle (217,174 163x49), "Hết ca", invisible if: not hienthiDialog2, input disabled if: not hienthiDialog2
            OnMouseDown: execute { bShift_is_over2 := TRUE; hienthiDialog2 := FALSE; }
    Rectangle (235,423 700x105), "WARNING: %s", text variable: StWarningTxt3, invisible if: not bAlarm_Iot, input disabled if: not bAlarm_Iot
END_VISUALIZATION

// ---- VISUs/Manual/Line1/N_FoodSupply1.TcVIS
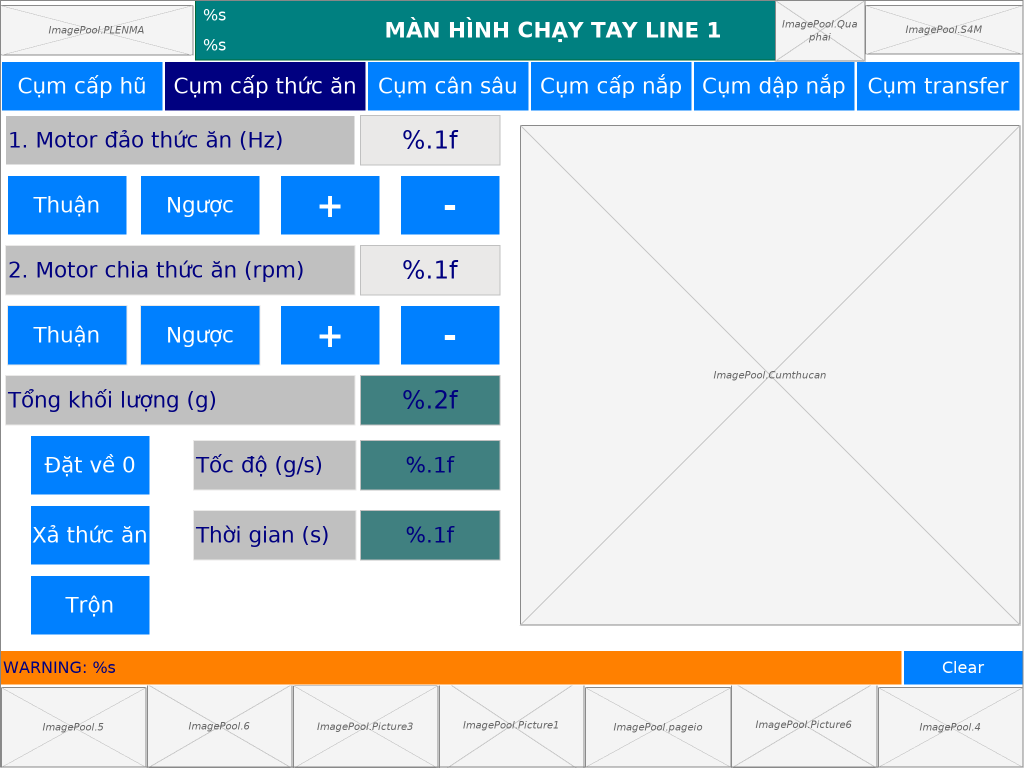
VISUALIZATION N_FoodSupply1  // 1024x768
    Rectangle (30,575 120x60), "Dừng", invisible if: not PR_Line01.daothucan, input disabled if: not PR_Line01.daothucan
        OnMouseDown: execute { PR_Line01.daothucan := FALSE; PR_Line01.bxa := true; }
    Rectangle (30,575 120x60), "Trộn", invisible if: PR_Line01.daothucan, input disabled if: PR_Line01.daothucan
        OnMouseDown: execute { PR_Line01.daothucan := TRUE; PR_Line01.bxa := TRUE; }
    Rectangle (140,175 120x60), "Dừng", invisible if: not PR_Line01.bMotor_mixer_reverse, input disabled if: not PR_Line01.bMotor_mixer_reverse
        OnMouseDown: execute { PR_Line01.bMotor_mixer_reverse := FALSE; }
    Rectangle (140,305 120x60), "Dừng", invisible if: not PR_Line01.bMotor_Food_reverse, input disabled if: not PR_Line01.bMotor_Food_reverse
        OnMouseDown: execute { PR_Line01.bMotor_Food_reverse := FALSE; PR_Line01.bxa := FALSE; }
    Rectangle (140,305 120x60), "Ngược", invisible if: PR_Line01.bMotor_Food_reverse, input disabled if: PR_Line01.bMotor_Food
        OnMouseDown: execute { PR_Line01.bMotor_Food_reverse := TRUE; PR_Line01.bxa := false; }
    Rectangle (140,175 120x60), "Ngược", invisible if: PR_Line01.bMotor_mixer_reverse, input disabled if: PR_Line01.bMotor_mixer_Manual
        OnMouseDown: execute { PR_Line01.bMotor_mixer_reverse := TRUE; PR_Line01.bxa := false; }
    Rectangle (7,305 120x60), "Dừng", invisible if: not PR_Line01.bMotor_Food, input disabled if: not PR_Line01.bMotor_Food
        OnMouseDown: execute { PR_Line01.bMotor_Food := FALSE; PR_Line01.bxa := FALSE; }
    Rectangle (7,305 120x60), "Thuận", invisible if: PR_Line01.bMotor_Food, input disabled if: PR_Line01.bMotor_Food_reverse
        OnMouseDown: execute { PR_Line01.bMotor_Food := TRUE; PR_Line01.bxa := false; }
    Rectangle (7,175 120x60), "Dừng", invisible if: not PR_Line01.bMotor_mixer_Manual, input disabled if: not PR_Line01.bMotor_mixer_Manual
        OnMouseDown: execute { PR_Line01.bMotor_mixer_Manual := FALSE; }
    Rectangle (7,175 120x60), "Thuận", invisible if: PR_Line01.bMotor_mixer_Manual, input disabled if: PR_Line01.bMotor_mixer_reverse
        OnMouseDown: execute { PR_Line01.bMotor_mixer_Manual := TRUE; PR_Line01.bxa := false; }
    Frame (0,687 1024x80)
        shows N_Footer_Line1()
    Frame (0,0 1024x60)
        shows N_Header()
    Textfield (353,5 400x50), "MÀN HÌNH CHẠY TAY LINE 1"
    Rectangle (5,115 350x50), "1. Motor đảo thức ăn (Hz)"
    Rectangle (5,245 350x50), "2. Motor chia thức ăn (rpm)"
    Rectangle (1,61 162x50), "Cụm cấp hũ"
        OnMouseClick: change screen: N_JarSupply1
    Rectangle (164,61 202x50), "Cụm cấp thức ăn"
        OnMouseClick: change screen: N_FoodSupply1
    Rectangle (367,61 162x50), "Cụm cân sâu"
        OnMouseClick: change screen: N_WormWeight1
    Rectangle (530,61 162x50), "Cụm cấp nắp"
        OnMouseClick: change screen: N_LidSupply1
    Rectangle (693,61 162x50), "Cụm dập nắp"
        OnMouseClick: change screen: N_LidPressing1
    Rectangle (856,61 164x50), "Cụm transfer"
        OnMouseClick: change screen: N_Tranfer1
    Rectangle (360,115 140x50), "%.1f", text variable: PR_Line01.fb_FoodMixer.fSpeed_motor_mixer_Manual
        OnMouseDown: write PR_Line01.fb_FoodMixer.fSpeed_motor_mixer_Manual via VisuDialogs.Numpad
    Rectangle (360,245 140x50), "%.1f", text variable: PR_Line01.fb_FoodWeight.fSpeed_Food_Motor_Manual
        OnMouseDown: write PR_Line01.fb_FoodWeight.fSpeed_Food_Motor_Manual via VisuDialogs.Numpad
    Rectangle (5,375 350x50), "Tổng khối lượng (g)"
    Rectangle (280,175 100x60), "+", colour toggle: PR_Line01.bUp_Motor_Mixer
        OnMouseDown: execute { PR_Line01.bUp_Motor_Mixer := TRUE; PR_Line01.bxa := false; }
    Rectangle (400,175 100x60), "-", colour toggle: PR_Line01.bDown_Motor_Mixer
        OnMouseDown: execute { PR_Line01.bDown_Motor_Mixer := TRUE; PR_Line01.bxa := false; }
    Rectangle (280,305 100x60), "+", colour toggle: PR_Line01.bUp_Food_Motor
        OnMouseDown: execute { PR_Line01.bUp_Food_Motor := TRUE; PR_Line01.bxa := FALSE; }
    Rectangle (400,305 100x60), "-", colour toggle: PR_Line01.bDown_Food_Motor
        OnMouseDown: execute { PR_Line01.bDown_Food_Motor := TRUE; PR_Line01.bxa := false; }
    Rectangle (360,375 140x50), "%.2f", text variable: PR_Line01.fb_FoodWeight.fWeight_Food
    Rectangle (193,440 163x50), "Tốc độ (g/s)"
    Rectangle (360,440 140x50), "%.1f", text variable: PR_Line01.fb_FoodWeight.fFlow_Food
    Image (775,0 90x61), input disabled if: bResetAuto2, image: ImagePool.Qua phai
        OnMouseClick: change screen: N_FoodSupply2
        OnMouseClick: execute { MAIN_LINE2.bModeManual := TRUE; MAIN_LINE2.bModeAuto := FALSE; }
    Rectangle (30,435 120x60), "Đặt về 0", colour toggle: PR_Line01.bZero_Loadcell_Food
        tap PR_Line01.bZero_Loadcell_Food
        OnMouseDown: execute { PR_Line01.bxa := false; }
        OnMouseUp: execute { PR_Line01.bZero_Loadcell_Food := TRUE; }
    Rectangle (30,505 120x60), "Xả thức ăn", colour toggle: PR_Line01.xathucan
        OnMouseDown: execute { PR_Line01.xathucan := TRUE; PR_Line01.bxa := TRUE; }
    Rectangle (193,510 163x50), "Thời gian (s)"
    Rectangle (360,510 140x50), "%.1f", text variable: PR_Line01.fb_FoodWeight.fTime
    Image (520,125 500x500), image: ImagePool.Cumthucan
    Frame (0,650 1024x35)
        shows N_Footer_Alarm()
END_VISUALIZATION

// ---- VISUs/Manual/Line1/N_JarSupply1.TcVIS
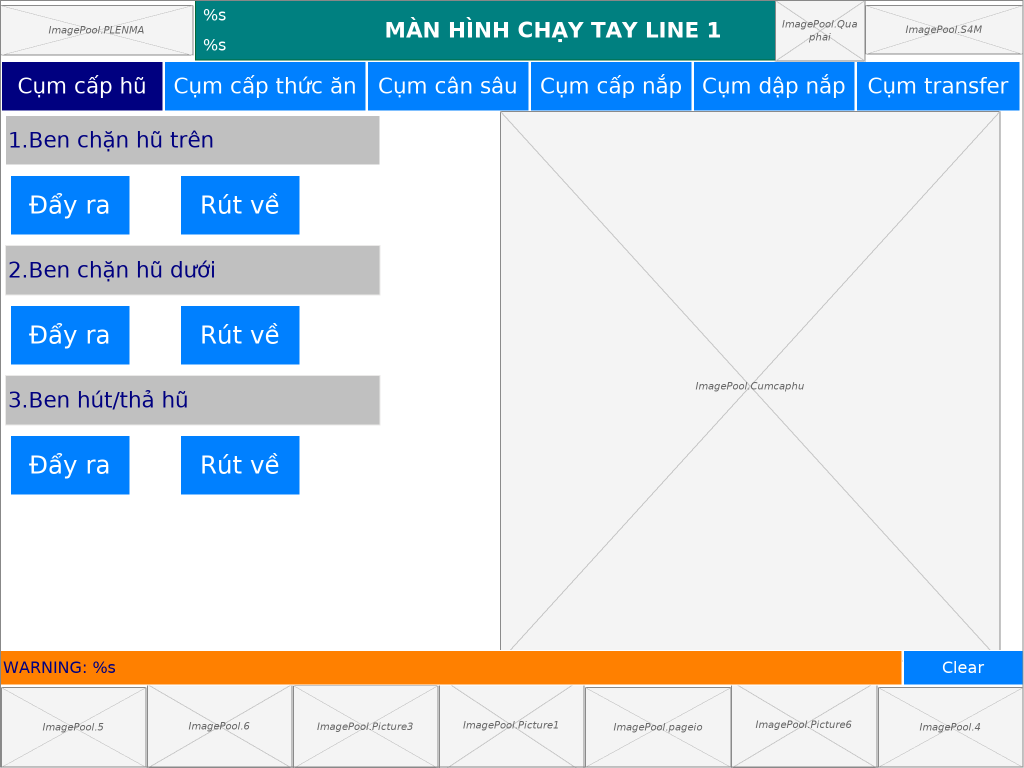
VISUALIZATION N_JarSupply1  // 1024x768
    Rectangle (10,305 120x60), "Đẩy ra", colour toggle: PR_Line01.bCylinder_dw_extend
        OnMouseDown: execute { PR_Line01.bCylinder_dw_extend := TRUE; PR_Line01.bCylinder_dw_retract := FALSE; }
    Rectangle (180,175 120x60), "Rút về", colour toggle: PR_Line01.bCylinder_up_retract
        OnMouseDown: execute { PR_Line01.bCylinder_up_retract := TRUE; PR_Line01.bCylinder_up_extend := FALSE; }
    Rectangle (180,305 120x60), "Rút về", colour toggle: PR_Line01.bCylinder_dw_retract
        OnMouseDown: execute { PR_Line01.bCylinder_dw_retract := TRUE; PR_Line01.bCylinder_dw_extend := FALSE; }
    Frame (0,687 1024x80)
        shows N_Footer_Line1()
    Frame (0,0 1024x60)
        shows N_Header()
    Textfield (353,5 400x50), "MÀN HÌNH CHẠY TAY LINE 1"
    Rectangle (5,115 375x50), "1.Ben chặn hũ trên"
    Rectangle (10,175 120x60), "Đẩy ra", colour toggle: PR_Line01.bCylinder_up_extend
        OnMouseDown: execute { PR_Line01.bCylinder_up_extend := TRUE; PR_Line01.bCylinder_up_retract := FALSE; }
    Rectangle (5,245 375x50), "2.Ben chặn hũ dưới"
    Rectangle (1,61 162x50), "Cụm cấp hũ"
        OnMouseClick: change screen: N_JarSupply1
    Rectangle (164,61 202x50), "Cụm cấp thức ăn"
        OnMouseClick: change screen: N_FoodSupply1
    Rectangle (367,61 162x50), "Cụm cân sâu"
        OnMouseClick: change screen: N_WormWeight1
    Rectangle (530,61 162x50), "Cụm cấp nắp"
        OnMouseClick: change screen: N_LidSupply1
    Rectangle (693,61 162x50), "Cụm dập nắp"
        OnMouseClick: change screen: N_LidPressing1
    Rectangle (856,61 164x50), "Cụm transfer"
        OnMouseClick: change screen: N_Tranfer1
    Image (775,0 90x61), input disabled if: bResetAuto2, image: ImagePool.Qua phai
        OnMouseClick: change screen: N_JarSupply2
        OnMouseClick: execute { MAIN_LINE2.bModeManual := TRUE; MAIN_LINE2.bModeAuto := FALSE; }
    Image (500,111 500x550), image: ImagePool.Cumcaphu
    Frame (0,650 1024x35)
        shows N_Footer_Alarm()
    Rectangle (10,435 120x60), "Đẩy ra", colour toggle: PR_Line01.bCylinder_Suction_cup_extend
        OnMouseDown: execute { PR_Line01.bCylinder_Suction_cup_extend := TRUE; PR_Line01.bCylinder_Suction_cup_retract := FALSE; }
    Rectangle (180,435 120x60), "Rút về", colour toggle: PR_Line01.bCylinder_Suction_cup_retract
        OnMouseDown: execute { PR_Line01.bCylinder_Suction_cup_extend := FALSE; PR_Line01.bCylinder_Suction_cup_retract := true; }
    Rectangle (5,375 375x50), "3.Ben hút/thả hũ"
END_VISUALIZATION

// ---- VISUs/Manual/Line1/N_LidPressing1.TcVIS
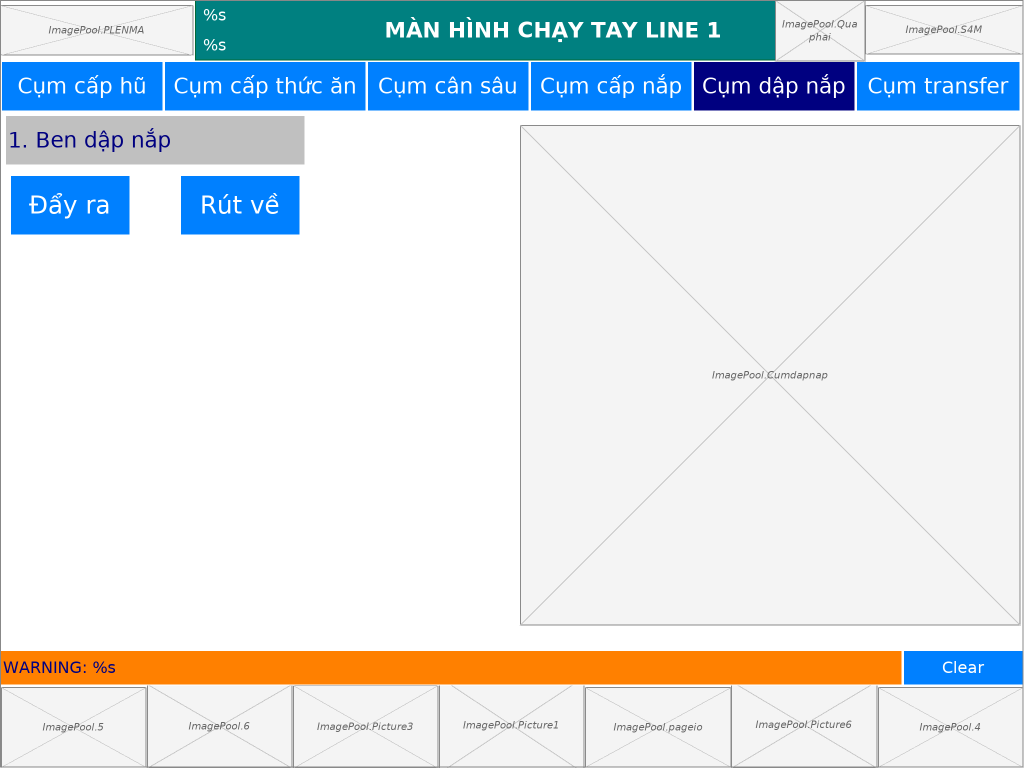
VISUALIZATION N_LidPressing1  // 1024x768
    Rectangle (180,175 120x60), "Rút về", colour toggle: PR_Line01.bCylinder_CloseLid_Retract
        OnMouseDown: execute { PR_Line01.bCylinder_CloseLid_Retract := TRUE; PR_Line01.bCylinder_CloseLid_Extend := FALSE; }
    Frame (0,687 1024x80)
        shows N_Footer_Line1()
    Frame (0,0 1024x60)
        shows N_Header()
    Textfield (353,5 400x50), "MÀN HÌNH CHẠY TAY LINE 1"
    Rectangle (5,115 300x50), "1. Ben dập nắp"
    Rectangle (10,175 120x60), "Đẩy ra", colour toggle: PR_Line01.bCylinder_CloseLid_Extend
        OnMouseDown: execute { PR_Line01.bCylinder_CloseLid_Extend := TRUE; PR_Line01.bCylinder_CloseLid_Retract := FALSE; }
    Rectangle (1,61 162x50), "Cụm cấp hũ"
        OnMouseClick: change screen: N_JarSupply1
    Rectangle (164,61 202x50), "Cụm cấp thức ăn"
        OnMouseClick: change screen: N_FoodSupply1
    Rectangle (367,61 162x50), "Cụm cân sâu"
        OnMouseClick: change screen: N_WormWeight1
    Rectangle (530,61 162x50), "Cụm cấp nắp"
        OnMouseClick: change screen: N_LidSupply1
    Rectangle (693,61 162x50), "Cụm dập nắp"
        OnMouseClick: change screen: N_LidPressing1
    Rectangle (856,61 164x50), "Cụm transfer"
        OnMouseClick: change screen: N_Tranfer1
    Image (775,0 90x61), input disabled if: bResetAuto2, image: ImagePool.Qua phai
        OnMouseClick: change screen: N_LidPressing2
        OnMouseClick: execute { MAIN_LINE2.bModeManual := TRUE; MAIN_LINE2.bModeAuto := FALSE; }
    Image (520,125 500x500), image: ImagePool.Cumdapnap
    Frame (0,650 1024x35)
        shows N_Footer_Alarm()
END_VISUALIZATION

// ---- VISUs/Manual/Line1/N_LidSupply1.TcVIS
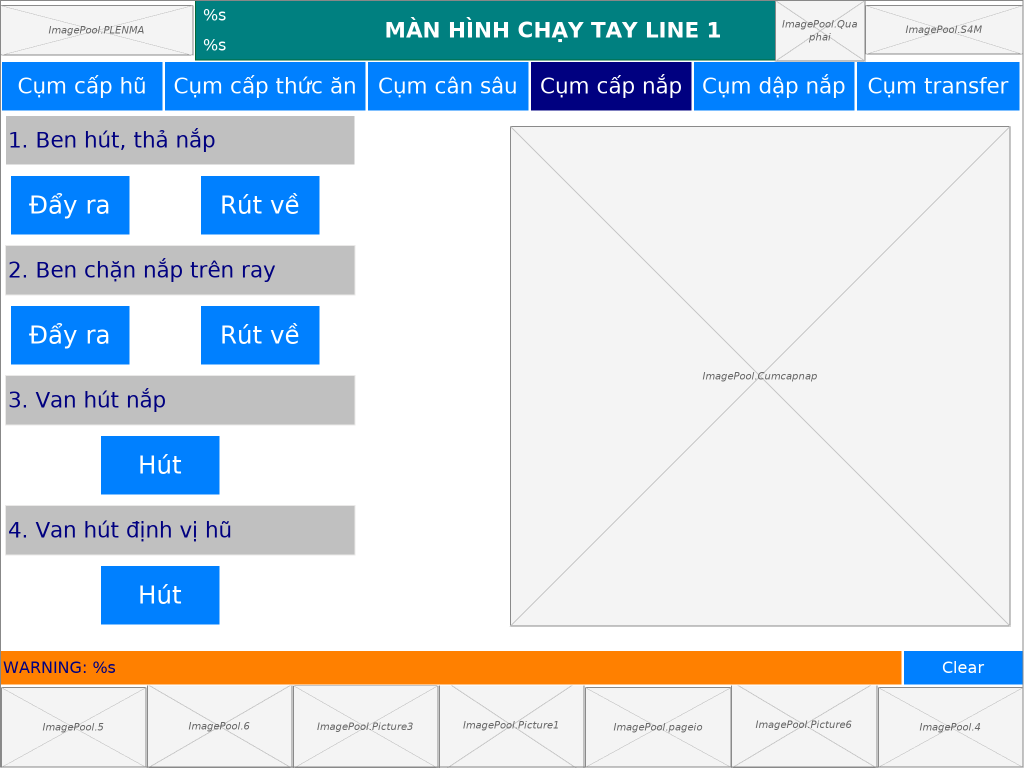
VISUALIZATION N_LidSupply1  // 1024x768
    Rectangle (100,565 120x60), "Dừng hút", invisible if: NOT PR_Line01.bCupSuctionValve, input disabled if: NOT PR_Line01.bCupSuctionValve
        OnMouseDown: execute { PR_Line01.bCupSuctionValve := false; }
    Rectangle (100,435 120x60), "Dừng hút", invisible if: not PR_Line01.bLidSuctionValve, input disabled if: not PR_Line01.bLidSuctionValve
        OnMouseDown: execute { PR_Line01.bLidSuctionValve := FALSE; }
    Rectangle (10,305 120x60), "Đẩy ra", colour toggle: PR_Line01.bCylinder_LidStopper_extend
        OnMouseDown: execute { PR_Line01.bCylinder_LidStopper_extend := TRUE; PR_Line01.bCylinder_LidStopper_retract := FALSE; }
    Rectangle (10,175 120x60), "Đẩy ra", colour toggle: PR_Line01.bCylinder_Suction_extend
        OnMouseDown: execute { PR_Line01.bCylinder_Suction_extend := TRUE; PR_Line01.bCylinder_Suction_retract := FALSE; }
    Rectangle (200,305 120x60), "Rút về", colour toggle: PR_Line01.bCylinder_LidStopper_retract
        OnMouseDown: execute { PR_Line01.bCylinder_LidStopper_retract := TRUE; PR_Line01.bCylinder_LidStopper_extend := FALSE; }
    Frame (0,687 1024x80)
        shows N_Footer_Line1()
    Frame (0,0 1024x60)
        shows N_Header()
    Textfield (353,5 400x50), "MÀN HÌNH CHẠY TAY LINE 1"
    Rectangle (5,115 350x50), "1. Ben hút, thả nắp"
    Rectangle (200,175 120x60), "Rút về", colour toggle: PR_Line01.bCylinder_Suction_retract
        toggle GVL_OF_VU.bValveBlowLid[1]
        OnMouseDown: execute { PR_Line01.bCylinder_Suction_retract := TRUE; PR_Line01.bCylinder_Suction_extend := FALSE; }
    Rectangle (5,245 350x50), "2. Ben chặn nắp trên ray"
    Rectangle (1,61 162x50), "Cụm cấp hũ"
        OnMouseClick: change screen: N_JarSupply1
    Rectangle (164,61 202x50), "Cụm cấp thức ăn"
        OnMouseClick: change screen: N_FoodSupply1
    Rectangle (367,61 162x50), "Cụm cân sâu"
        OnMouseClick: change screen: N_WormWeight1
    Rectangle (530,61 162x50), "Cụm cấp nắp"
        OnMouseClick: change screen: N_LidSupply1
    Rectangle (693,61 162x50), "Cụm dập nắp"
        OnMouseClick: change screen: N_LidPressing1
    Rectangle (856,61 164x50), "Cụm transfer"
        OnMouseClick: change screen: N_Tranfer1
    Rectangle (5,375 350x50), "3. Van hút nắp"
    Rectangle (100,435 120x60), "Hút", invisible if: PR_Line01.bLidSuctionValve, input disabled if: PR_Line01.bLidSuctionValve
        OnMouseDown: execute { PR_Line01.bLidSuctionValve := TRUE; }
    Image (775,0 90x61), input disabled if: bResetAuto2, image: ImagePool.Qua phai
        OnMouseClick: change screen: N_LidSupply2
        OnMouseClick: execute { MAIN_LINE2.bModeManual := TRUE; MAIN_LINE2.bModeAuto := FALSE; }
    Rectangle (5,505 350x50), "4. Van hút định vị hũ"
    Rectangle (100,565 120x60), "Hút", invisible if: PR_Line01.bCupSuctionValve, input disabled if: PR_Line01.bCupSuctionValve
        OnMouseDown: execute { PR_Line01.bCupSuctionValve := true; }
    Image (510,126 500x500), image: ImagePool.Cumcapnap
    Frame (0,650 1024x35)
        shows N_Footer_Alarm()
END_VISUALIZATION

// ---- VISUs/Manual/Line1/N_Tranfer1.TcVIS
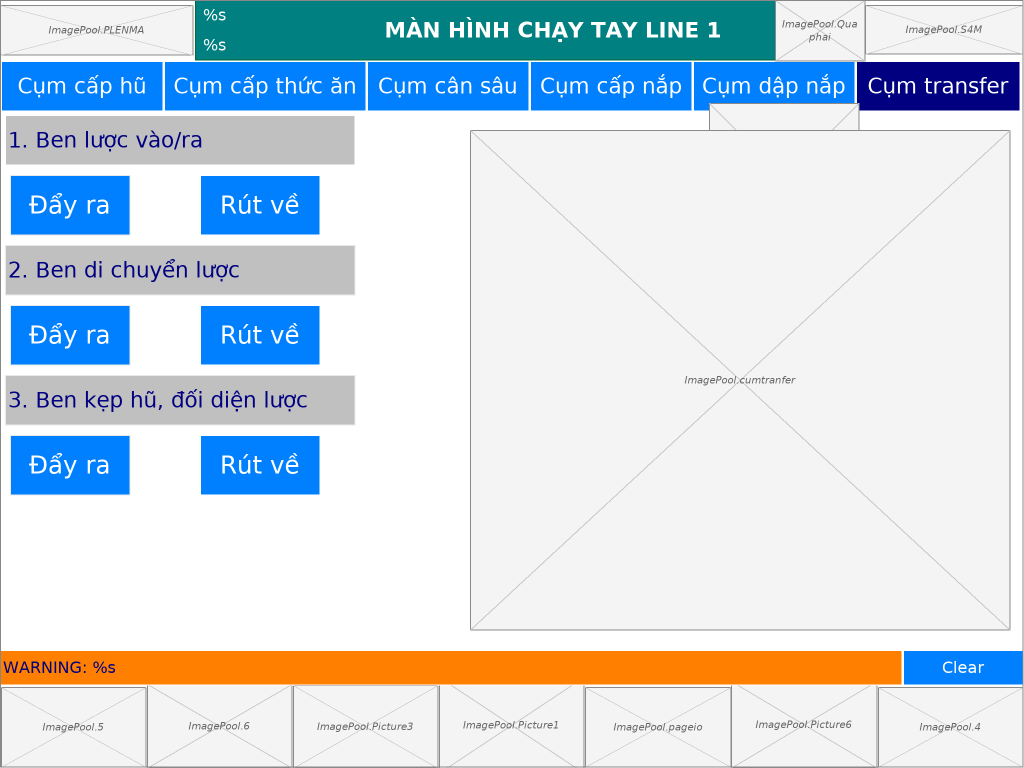
VISUALIZATION N_Tranfer1  // 1024x768
    Rectangle (10,305 120x60), "Đẩy ra", colour toggle: PR_Line01.bCylinder_Move_Comb_Extend, input disabled if: Not PR_Line01.bCheck
        OnMouseDown: execute {
            PR_Line01.bCylinder_Move_Comb_Extend := TRUE;
            PR_Line01.bCylinder_Move_Comb_Retract := FALSE;
            PR_Line01.bxa := FALSE;
        }
    Rectangle (200,175 120x60), "Rút về", colour toggle: PR_Line01.bCylinder_Comb_Retract
        OnMouseDown: execute {
            PR_Line01.bCylinder_Comb_Retract := TRUE;
            PR_Line01.bCylinder_Comb_Extend := FALSE;
            PR_Line01.bxa := FALSE;
        }
    Rectangle (200,305 120x60), "Rút về", colour toggle: PR_Line01.bCylinder_Move_Comb_Retract, input disabled if: Not PR_Line01.bCheck
        OnMouseDown: execute {
            PR_Line01.bCylinder_Move_Comb_Retract := TRUE;
            PR_Line01.bCylinder_Move_Comb_Extend := FALSE;
            PR_Line01.bxa := FALSE;
        }
    Frame (0,687 1024x80)
        shows N_Footer_Line1()
    Frame (0,0 1024x60)
        shows N_Header()
    Textfield (353,5 400x50), "MÀN HÌNH CHẠY TAY LINE 1"
    Rectangle (5,115 350x50), "1. Ben lược vào/ra"
    Rectangle (10,175 120x60), "Đẩy ra", colour toggle: PR_Line01.bCylinder_Comb_Extend, input disabled if: Not PR_Line01.bCheck
        OnMouseDown: execute {
            PR_Line01.bCylinder_Comb_Extend := TRUE;
            PR_Line01.bCylinder_Comb_Retract := FALSE;
            PR_Line01.bxa := FALSE;
        }
    Rectangle (5,245 350x50), "2. Ben di chuyển lược"
    Rectangle (1,61 162x50), "Cụm cấp hũ"
        OnMouseClick: change screen: N_JarSupply1
    Rectangle (164,61 202x50), "Cụm cấp thức ăn"
        OnMouseClick: change screen: N_FoodSupply1
    Rectangle (367,61 162x50), "Cụm cân sâu"
        OnMouseClick: change screen: N_WormWeight1
    Rectangle (530,61 162x50), "Cụm cấp nắp"
        OnMouseClick: change screen: N_LidSupply1
    Rectangle (693,61 162x50), "Cụm dập nắp"
        OnMouseClick: change screen: N_LidPressing1
    Rectangle (856,61 164x50), "Cụm transfer"
        OnMouseClick: change screen: N_Tranfer1
    Rectangle (5,375 350x50), "3. Ben kẹp hũ, đối diện lược"
    Rectangle (200,435 120x60), "Rút về", text variable: GVL_OF_VU.fFreqOutputConveyor, colour toggle: PR_Line01.bCylinder_Clip_Retract
        OnMouseDown: execute {
            PR_Line01.bCylinder_Clip_Retract := TRUE;
            PR_Line01.bCylinder_Clip_Extend := FALSE;
            PR_Line01.bxa := FALSE;
        }
    Rectangle (10,435 120x60), "Đẩy ra", colour toggle: PR_Line01.bCylinder_Clip_Extend
        OnMouseDown: execute {
            PR_Line01.bCylinder_Clip_Extend := TRUE;
            PR_Line01.bCylinder_Clip_Retract := FALSE;
            PR_Line01.bxa := FALSE;
        }
    Image (709,103 150x150)
    Image (775,0 90x61), image: ImagePool.Qua phai
        OnMouseClick: change screen: N_Tranfer2
        OnMouseClick: execute { MAIN_LINE2.bModeManual := TRUE; MAIN_LINE2.bModeAuto := FALSE; }
    Image (470,130 540x500), image: ImagePool.cumtranfer
    Frame (0,650 1024x35)
        shows N_Footer_Alarm()
END_VISUALIZATION

// ---- VISUs/Manual/Line1/N_WormWeight1.TcVIS
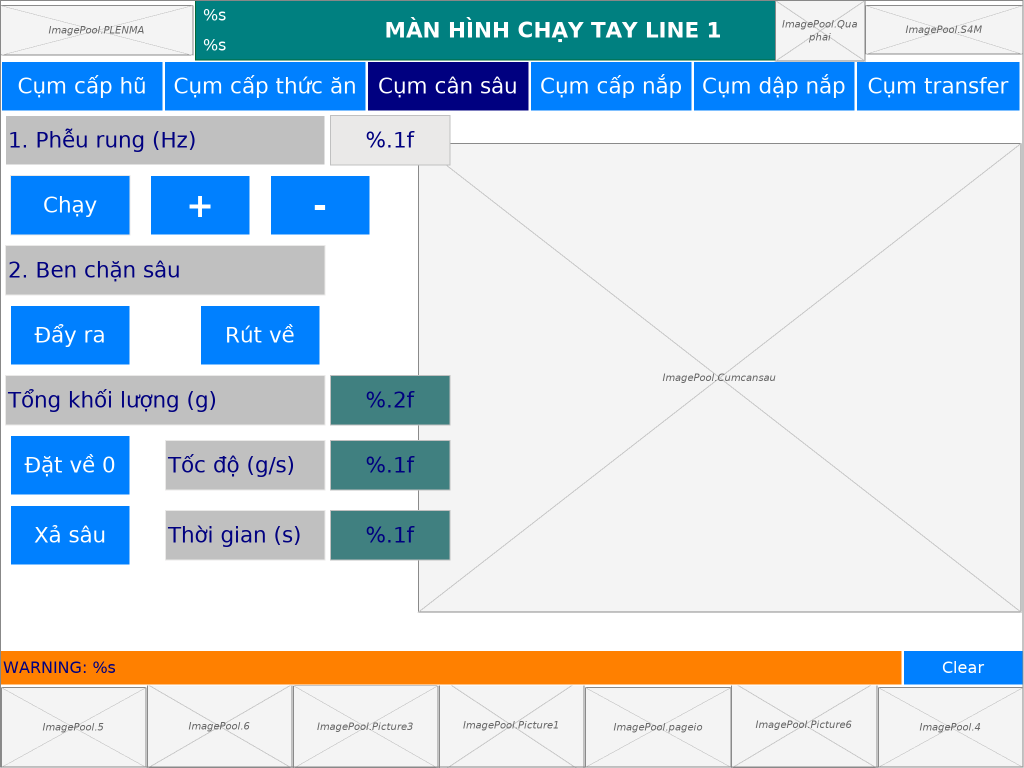
VISUALIZATION N_WormWeight1  // 1024x768
    Image (418,143 603x469), image: ImagePool.Cumcansau
    Rectangle (10,175 120x60), "Dừng", invisible if: not PR_Line01.bMotor_vibrating_funnel, input disabled if: not PR_Line01.bMotor_vibrating_funnel
        OnMouseDown: execute { PR_Line01.bMotor_vibrating_funnel := FALSE; PR_Line01.bxa := FALSE; }
    Rectangle (10,175 120x60), "Chạy", invisible if: PR_Line01.bMotor_vibrating_funnel, input disabled if: PR_Line01.bMotor_vibrating_funnel
        OnMouseDown: execute { PR_Line01.bMotor_vibrating_funnel := TRUE; PR_Line01.bxa := FALSE; }
    Rectangle (10,305 120x60), "Đẩy ra", colour toggle: PR_Line01.bCylinder_Block_Worm_Extend
        OnMouseDown: execute {
            PR_Line01.bCylinder_Block_Worm_Extend := TRUE;
            PR_Line01.bCylinder_Block_Worm_Retract := FALSE;
            PR_Line01.bxa := FALSE;
        }
    Rectangle (200,305 120x60), "Rút về", colour toggle: PR_Line01.bCylinder_Block_Worm_Retract
        OnMouseDown: execute {
            PR_Line01.bCylinder_Block_Worm_Retract := TRUE;
            PR_Line01.bCylinder_Block_Worm_Extend := FALSE;
            PR_Line01.bxa := FALSE;
        }
    Frame (0,687 1024x80)
        shows N_Footer_Line1()
    Frame (0,0 1024x60)
        shows N_Header()
    Textfield (353,5 400x50), "MÀN HÌNH CHẠY TAY LINE 1"
    Rectangle (5,115 320x50), "1. Phễu rung (Hz)"
    Rectangle (5,245 320x50), "2. Ben chặn sâu"
    Rectangle (1,61 162x50), "Cụm cấp hũ"
        OnMouseClick: change screen: N_JarSupply1
    Rectangle (164,61 202x50), "Cụm cấp thức ăn"
        OnMouseClick: change screen: N_FoodSupply1
    Rectangle (367,61 162x50), "Cụm cân sâu"
        OnMouseClick: change screen: N_WormWeight1
    Rectangle (530,61 162x50), "Cụm cấp nắp"
        OnMouseClick: change screen: N_LidSupply1
    Rectangle (693,61 162x50), "Cụm dập nắp"
        OnMouseClick: change screen: N_LidPressing1
    Rectangle (856,61 164x50), "Cụm transfer"
        OnMouseClick: change screen: N_Tranfer1
    Rectangle (330,115 120x50), "%.1f", text variable: PR_Line01.fb_WormWeight.fSpeed_vibrating_funnel_Manual
        OnMouseDown: write PR_Line01.fb_WormWeight.fSpeed_vibrating_funnel_Manual via VisuDialogs.Numpad
        OnMouseDown: execute { PR_Line01.bxa := FALSE; }
    Rectangle (5,375 320x50), "Tổng khối lượng (g)"
    Rectangle (150,175 100x60), "+", colour toggle: PR_Line01.bUp_vibrating_funnel
        OnMouseDown: execute { PR_Line01.bUp_vibrating_funnel := TRUE; PR_Line01.bxa := FALSE; }
    Rectangle (270,175 100x60), "-", colour toggle: PR_Line01.bDown_vibrating_funnel
        OnMouseDown: execute { PR_Line01.bDown_vibrating_funnel := TRUE; PR_Line01.bxa := FALSE; }
    Rectangle (330,375 120x50), "%.2f", text variable: PR_Line01.fb_WormWeight.fWeight_Worm
    Rectangle (10,435 120x60), "Đặt về 0"
        tap PR_Line01.bZero_Loadcell_Worm
        OnMouseDown: execute { PR_Line01.bxa := FALSE; }
        OnMouseUp: execute { PR_Line01.bZero_Loadcell_Worm := TRUE; }
    Rectangle (165,440 160x50), "Tốc độ (g/s)"
    Rectangle (330,440 120x50), "%.1f", text variable: PR_Line01.fb_WormWeight.fFlow_Worm
    Image (775,0 90x61), input disabled if: bResetAuto2, image: ImagePool.Qua phai
        OnMouseClick: change screen: N_WormWeight2
        OnMouseClick: execute { MAIN_LINE2.bModeManual := TRUE; MAIN_LINE2.bModeAuto := FALSE; }
    Rectangle (10,505 120x60), "Xả sâu", colour toggle: PR_Line01.xasau
        OnMouseDown: execute { PR_Line01.xasau := TRUE; PR_Line01.bxa := true; }
    Rectangle (165,510 160x50), "Thời gian (s)"
    Rectangle (330,510 120x50), "%.1f", text variable: PR_Line01.fb_WormWeight.fTime
    Frame (0,650 1024x35)
        shows N_Footer_Alarm()
END_VISUALIZATION

// ---- VISUs/Manual/Line2/N_FoodSupply2.TcVIS
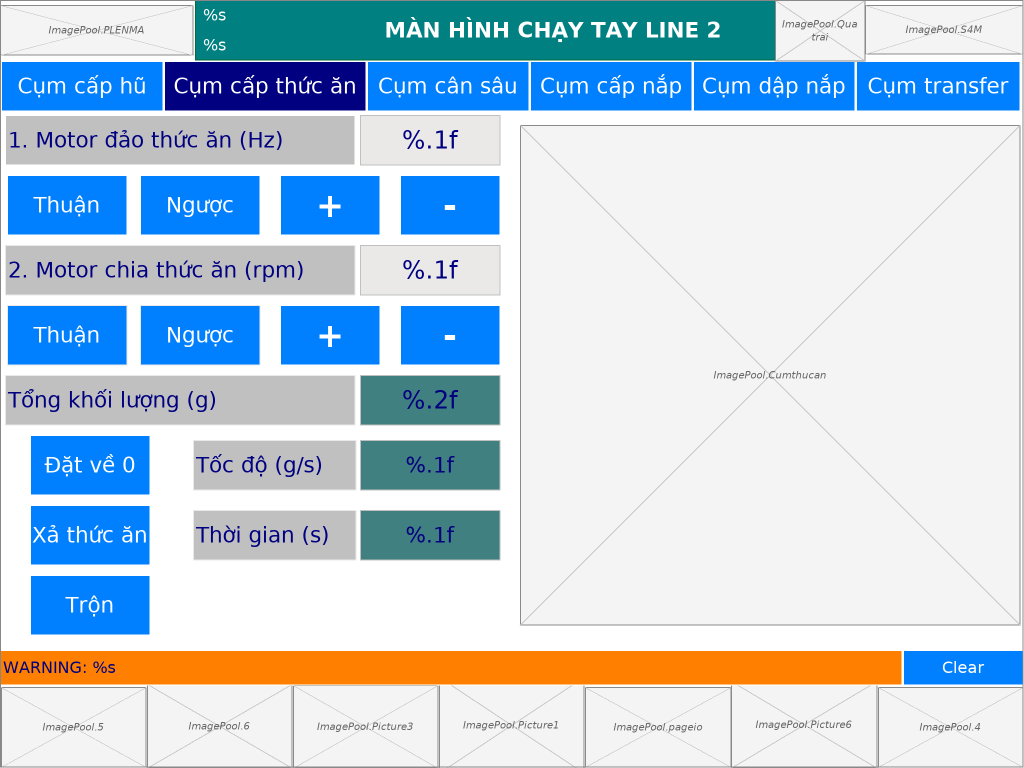
VISUALIZATION N_FoodSupply2  // 1024x768
    Rectangle (7,305 120x60), "Dừng", invisible if: not PR_Line02.bMotor_Food, input disabled if: not PR_Line02.bMotor_Food
        OnMouseDown: execute { PR_Line02.bMotor_Food := FALSE; PR_Line02.bxa := FALSE; }
    Rectangle (7,305 120x60), "Thuận", invisible if: PR_Line02.bMotor_Food, input disabled if: PR_Line02.bMotor_Food_reverse
        OnMouseDown: execute { PR_Line02.bMotor_Food := TRUE; PR_Line02.bxa := false; }
    Rectangle (140,305 120x60), "Dừng", invisible if: not PR_Line02.bMotor_Food_reverse, input disabled if: not PR_Line02.bMotor_Food_reverse
        OnMouseDown: execute { PR_Line02.bMotor_Food_reverse := FALSE; PR_Line02.bxa := FALSE; }
    Rectangle (140,305 120x60), "Ngược", invisible if: PR_Line02.bMotor_Food_reverse, input disabled if: PR_Line02.bMotor_Food
        OnMouseDown: execute { PR_Line02.bMotor_Food_reverse := TRUE; PR_Line02.bxa := false; }
    Rectangle (140,175 120x60), "Dừng", invisible if: not PR_Line02.bMotor_mixer_reverse, input disabled if: not PR_Line02.bMotor_mixer_reverse
        OnMouseDown: execute { PR_Line02.bMotor_mixer_reverse := FALSE; }
    Rectangle (140,175 120x60), "Ngược", invisible if: PR_Line02.bMotor_mixer_reverse, input disabled if: PR_Line02.bMotor_mixer_Manual
        OnMouseDown: execute { PR_Line02.bMotor_mixer_reverse := TRUE; PR_Line02.bxa := false; }
    Rectangle (7,175 120x60), "Dừng", invisible if: not PR_Line02.bMotor_mixer_Manual, input disabled if: not PR_Line02.bMotor_mixer_Manual
        OnMouseDown: execute { PR_Line02.bMotor_mixer_Manual := FALSE; }
    Rectangle (7,175 120x60), "Thuận", invisible if: PR_Line02.bMotor_mixer_Manual, input disabled if: PR_Line02.bMotor_mixer_reverse
        OnMouseDown: execute { PR_Line02.bMotor_mixer_Manual := TRUE; PR_Line02.bxa := false; }
    Frame (0,687 1024x80)
        shows N_Footer_Line2()
    Frame (0,0 1024x60)
        shows N_Header()
    Textfield (353,5 400x50), "MÀN HÌNH CHẠY TAY LINE 2"
    Rectangle (1,61 162x50), "Cụm cấp hũ"
        OnMouseClick: change screen: N_JarSupply2
    Rectangle (164,61 202x50), "Cụm cấp thức ăn"
        OnMouseClick: change screen: N_FoodSupply2
    Rectangle (367,61 162x50), "Cụm cân sâu"
        OnMouseClick: change screen: N_WormWeight2
    Rectangle (530,61 162x50), "Cụm cấp nắp"
        OnMouseClick: change screen: N_LidSupply2
    Rectangle (693,61 162x50), "Cụm dập nắp"
        OnMouseClick: change screen: N_LidPressing2
    Rectangle (856,61 164x50), "Cụm transfer"
        OnMouseClick: change screen: N_Tranfer2
    Image (775,0 90x61), input disabled if: bResetAuto1, image: ImagePool.Qua trai
        OnMouseClick: change screen: N_FoodSupply1
        OnMouseClick: execute { MAIN.bModeManual := TRUE; MAIN.bModeAuto := FALSE; }
    Image (520,125 500x500), image: ImagePool.Cumthucan
    Rectangle (30,575 120x60), "Dừng", invisible if: not PR_Line02.daothucan, input disabled if: not PR_Line02.daothucan
        OnMouseDown: execute { PR_Line02.daothucan := FALSE; PR_Line02.bxa := true; }
    Rectangle (5,115 350x50), "1. Motor đảo thức ăn (Hz)"
    Rectangle (5,245 350x50), "2. Motor chia thức ăn (rpm)"
    Rectangle (360,115 140x50), "%.1f", text variable: PR_Line02.fb_FoodMixer.fSpeed_motor_mixer_Manual
        OnMouseDown: write PR_Line02.fb_FoodMixer.fSpeed_motor_mixer_Manual via VisuDialogs.Numpad
    Rectangle (360,245 140x50), "%.1f", text variable: PR_Line02.fb_FoodWeight.fSpeed_Food_Motor_Manual
        OnMouseDown: write PR_Line02.fb_FoodWeight.fSpeed_Food_Motor_Manual via VisuDialogs.Numpad
    Rectangle (5,375 350x50), "Tổng khối lượng (g)"
    Rectangle (280,175 100x60), "+", colour toggle: PR_Line02.bUp_Motor_Mixer
        OnMouseDown: execute { PR_Line02.bUp_Motor_Mixer := TRUE; PR_Line02.bxa := false; }
    Rectangle (400,175 100x60), "-", colour toggle: PR_Line02.bDown_Motor_Mixer
        OnMouseDown: execute { PR_Line02.bDown_Motor_Mixer := TRUE; PR_Line02.bxa := false; }
    Rectangle (280,305 100x60), "+", colour toggle: PR_Line02.bUp_Food_Motor
        OnMouseDown: execute { PR_Line02.bUp_Food_Motor := TRUE; PR_Line02.bxa := FALSE; }
    Rectangle (400,305 100x60), "-", colour toggle: PR_Line02.bDown_Food_Motor
        OnMouseDown: execute { PR_Line02.bDown_Food_Motor := TRUE; PR_Line02.bxa := false; }
    Rectangle (360,375 140x50), "%.2f", text variable: PR_Line02.fb_FoodWeight.fWeight_Food
    Rectangle (193,440 163x50), "Tốc độ (g/s)"
    Rectangle (360,440 140x50), "%.1f", text variable: PR_Line02.fb_FoodWeight.fFlow_Food
    Rectangle (30,435 120x60), "Đặt về 0", colour toggle: PR_Line02.bZero_Loadcell_Food
        tap PR_Line02.bZero_Loadcell_Food p1329445385=TRUE
        OnMouseDown: execute { PR_Line02.bxa := false; }
        OnMouseUp: execute { PR_Line02.bZero_Loadcell_Food := TRUE; }
    Rectangle (30,505 120x60), "Xả thức ăn", colour toggle: PR_Line02.xathucan
        OnMouseDown: execute { PR_Line02.xathucan := TRUE; PR_Line02.bxa := TRUE; }
    Rectangle (193,510 163x50), "Thời gian (s)"
    Rectangle (360,510 140x50), "%.1f", text variable: PR_Line02.fb_FoodWeight.fTime
    Rectangle (30,575 120x60), "Trộn", invisible if: PR_Line02.daothucan, input disabled if: PR_Line02.daothucan
        OnMouseDown: execute { PR_Line02.daothucan := TRUE; PR_Line02.bxa := TRUE; }
    Frame (0,650 1024x35)
        shows N_Footer_Alarm_1()
END_VISUALIZATION

// ---- VISUs/Manual/Line2/N_JarSupply2.TcVIS
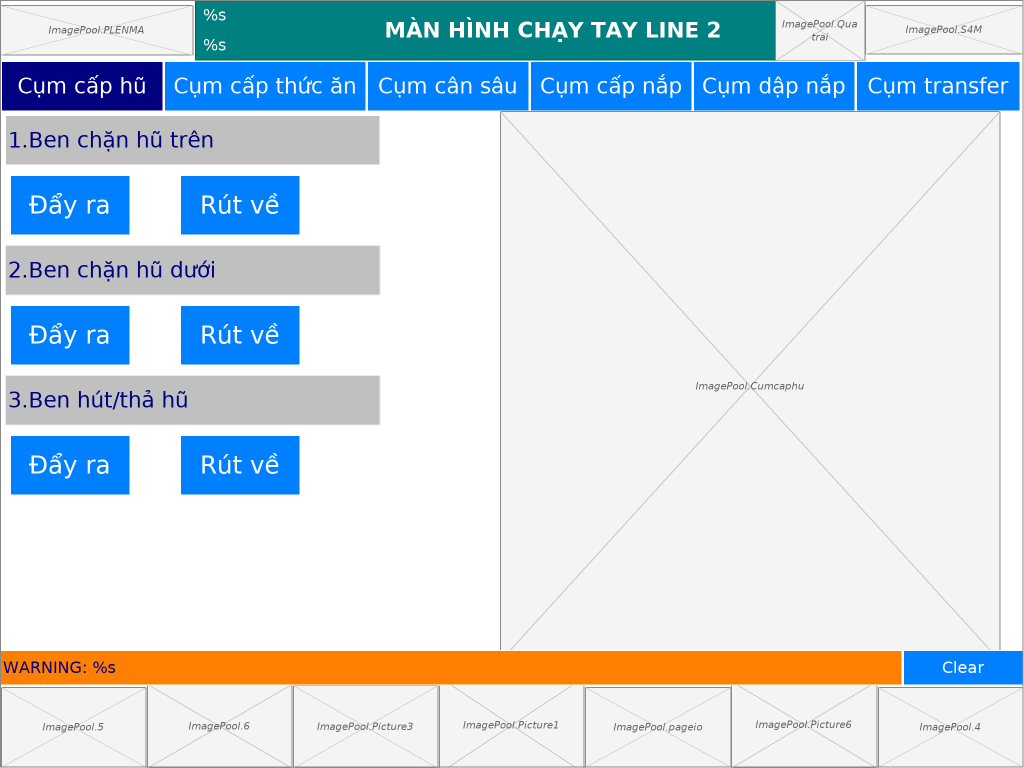
VISUALIZATION N_JarSupply2  // 1024x768
    Rectangle (10,305 120x60), "Đẩy ra", colour toggle: PR_Line02.bCylinder_dw_extend
        OnMouseDown: execute { PR_Line02.bCylinder_dw_extend := TRUE; PR_Line02.bCylinder_dw_retract := FALSE; }
    Rectangle (180,175 120x60), "Rút về", colour toggle: PR_Line02.bCylinder_up_retract
        OnMouseDown: execute { PR_Line02.bCylinder_up_retract := TRUE; PR_Line02.bCylinder_up_extend := FALSE; }
    Rectangle (180,305 120x60), "Rút về", colour toggle: PR_Line02.bCylinder_dw_retract
        OnMouseDown: execute { PR_Line02.bCylinder_dw_retract := TRUE; PR_Line02.bCylinder_dw_extend := FALSE; }
    Frame (0,687 1024x80)
        shows N_Footer_Line2()
    Frame (0,0 1024x60)
        shows N_Header()
    Textfield (353,5 400x50), "MÀN HÌNH CHẠY TAY LINE 2"
    Rectangle (10,175 120x60), "Đẩy ra", colour toggle: PR_Line02.bCylinder_up_extend
        OnMouseDown: execute { PR_Line02.bCylinder_up_extend := TRUE; PR_Line02.bCylinder_up_retract := FALSE; }
    Image (775,0 90x61), input disabled if: bResetAuto1, image: ImagePool.Qua trai
        OnMouseClick: change screen: N_JarSupply1
        OnMouseClick: execute { MAIN.bModeManual := TRUE; MAIN.bModeAuto := FALSE; }
    Rectangle (1,61 162x50), "Cụm cấp hũ"
        OnMouseClick: change screen: N_JarSupply2
    Rectangle (164,61 202x50), "Cụm cấp thức ăn"
        OnMouseClick: change screen: N_FoodSupply2
    Rectangle (367,61 162x50), "Cụm cân sâu"
        OnMouseClick: change screen: N_WormWeight2
    Rectangle (530,61 162x50), "Cụm cấp nắp"
        OnMouseClick: change screen: N_LidSupply2
    Rectangle (693,61 162x50), "Cụm dập nắp"
        OnMouseClick: change screen: N_LidPressing2
    Rectangle (856,61 164x50), "Cụm transfer"
        OnMouseClick: change screen: N_Tranfer2
    Rectangle (5,115 375x50), "1.Ben chặn hũ trên"
    Rectangle (5,245 375x50), "2.Ben chặn hũ dưới"
    Image (500,111 500x550), image: ImagePool.Cumcaphu
    Frame (0,650 1024x35)
        shows N_Footer_Alarm()
    Rectangle (10,435 120x60), "Đẩy ra", colour toggle: PR_Line02.bCylinder_Suction_cup_extend
        OnMouseDown: execute { PR_Line02.bCylinder_Suction_cup_extend := TRUE; PR_Line02.bCylinder_Suction_cup_retract := FALSE; }
    Rectangle (180,435 120x60), "Rút về", colour toggle: PR_Line02.bCylinder_Suction_cup_retract
        OnMouseDown: execute { PR_Line02.bCylinder_Suction_cup_extend := FALSE; PR_Line02.bCylinder_Suction_cup_retract := true; }
    Rectangle (5,375 375x50), "3.Ben hút/thả hũ"
END_VISUALIZATION

// ---- VISUs/Manual/Line2/N_LidPressing2.TcVIS
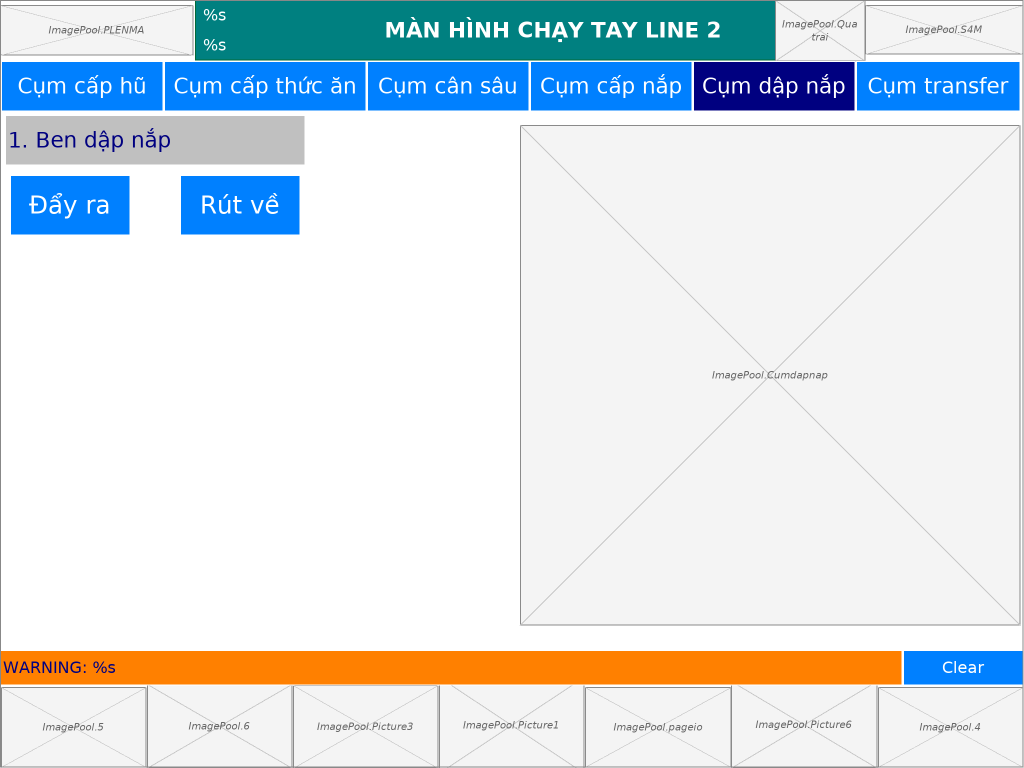
VISUALIZATION N_LidPressing2  // 1024x768
    Rectangle (180,175 120x60), "Rút về", colour toggle: PR_Line02.bCylinder_CloseLid_Retract
        OnMouseDown: execute { PR_Line02.bCylinder_CloseLid_Retract := TRUE; PR_Line02.bCylinder_CloseLid_Extend := FALSE; }
    Frame (0,687 1024x80)
        shows N_Footer_Line2()
    Frame (0,0 1024x60)
        shows N_Header()
    Textfield (353,5 400x50), "MÀN HÌNH CHẠY TAY LINE 2"
    Rectangle (10,175 120x60), "Đẩy ra", colour toggle: PR_Line02.bCylinder_CloseLid_Extend
        OnMouseDown: execute { PR_Line02.bCylinder_CloseLid_Extend := TRUE; PR_Line02.bCylinder_CloseLid_Retract := FALSE; }
    Image (775,0 90x61), input disabled if: bResetAuto1, image: ImagePool.Qua trai
        OnMouseClick: change screen: N_LidPressing1
        OnMouseClick: execute { MAIN.bModeManual := TRUE; MAIN.bModeAuto := FALSE; }
    Rectangle (1,61 162x50), "Cụm cấp hũ"
        OnMouseClick: change screen: N_JarSupply2
    Rectangle (164,61 202x50), "Cụm cấp thức ăn"
        OnMouseClick: change screen: N_FoodSupply2
    Rectangle (367,61 162x50), "Cụm cân sâu"
        OnMouseClick: change screen: N_WormWeight2
    Rectangle (530,61 162x50), "Cụm cấp nắp"
        OnMouseClick: change screen: N_LidSupply2
    Rectangle (693,61 162x50), "Cụm dập nắp"
        OnMouseClick: change screen: N_LidPressing2
    Rectangle (856,61 164x50), "Cụm transfer"
        OnMouseClick: change screen: N_Tranfer2
    Image (520,125 500x500), image: ImagePool.Cumdapnap
    Rectangle (5,115 300x50), "1. Ben dập nắp"
    Frame (0,650 1024x35)
        shows N_Footer_Alarm()
END_VISUALIZATION

// ---- VISUs/Manual/Line2/N_LidSupply2.TcVIS
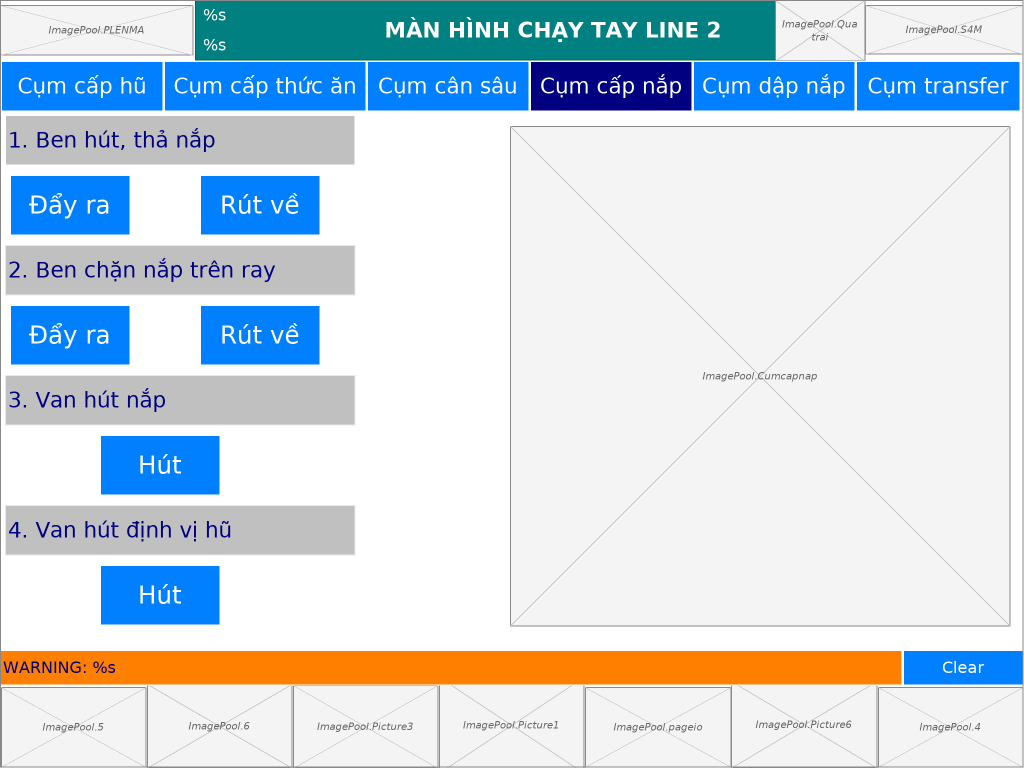
VISUALIZATION N_LidSupply2  // 1024x768
    Rectangle (10,305 120x60), "Đẩy ra", colour toggle: PR_Line02.bCylinder_LidStopper_extend
        OnMouseDown: execute { PR_Line02.bCylinder_LidStopper_extend := TRUE; PR_Line02.bCylinder_LidStopper_retract := FALSE; }
    Rectangle (200,175 120x60), "Rút về", colour toggle: PR_Line02.bCylinder_Suction_retract
        OnMouseDown: execute { PR_Line02.bCylinder_Suction_retract := TRUE; PR_Line02.bCylinder_Suction_extend := FALSE; }
    Rectangle (200,305 120x60), "Rút về", colour toggle: PR_Line02.bCylinder_LidStopper_retract
        OnMouseDown: execute { PR_Line02.bCylinder_LidStopper_retract := TRUE; PR_Line02.bCylinder_LidStopper_extend := FALSE; }
    Frame (0,687 1024x80)
        shows N_Footer_Line2()
    Frame (0,0 1024x60)
        shows N_Header()
    Textfield (353,5 400x50), "MÀN HÌNH CHẠY TAY LINE 2"
    Rectangle (10,175 120x60), "Đẩy ra", colour toggle: PR_Line02.bCylinder_Suction_extend
        OnMouseDown: execute { PR_Line02.bCylinder_Suction_extend := TRUE; PR_Line02.bCylinder_Suction_retract := FALSE; }
    Rectangle (100,435 120x60), "Dừng hút", invisible if: not PR_Line02.bLidSuctionValve, input disabled if: not PR_Line02.bLidSuctionValve
        OnMouseDown: execute { PR_Line02.bLidSuctionValve := FALSE; }
    Image (775,0 90x61), input disabled if: bResetAuto1, image: ImagePool.Qua trai
        OnMouseClick: change screen: N_LidSupply1
        OnMouseClick: execute { MAIN.bModeManual := TRUE; MAIN.bModeAuto := FALSE; }
    Rectangle (100,565 120x60), "Dừng hút", invisible if: not PR_Line02.bCupSuctionValve, input disabled if: not PR_Line02.bCupSuctionValve
        OnMouseDown: execute { PR_Line02.bCupSuctionValve := false; }
    Rectangle (1,61 162x50), "Cụm cấp hũ"
        OnMouseClick: change screen: N_JarSupply2
    Rectangle (164,61 202x50), "Cụm cấp thức ăn"
        OnMouseClick: change screen: N_FoodSupply2
    Rectangle (367,61 162x50), "Cụm cân sâu"
        OnMouseClick: change screen: N_WormWeight2
    Rectangle (530,61 162x50), "Cụm cấp nắp"
        OnMouseClick: change screen: N_LidSupply2
    Rectangle (693,61 162x50), "Cụm dập nắp"
        OnMouseClick: change screen: N_LidPressing2
    Rectangle (856,61 164x50), "Cụm transfer"
        OnMouseClick: change screen: N_Tranfer2
    Rectangle (100,435 120x60), "Hút", invisible if: PR_Line02.bLidSuctionValve, input disabled if: PR_Line02.bLidSuctionValve
        OnMouseDown: execute { PR_Line02.bLidSuctionValve := TRUE; }
    Rectangle (100,565 120x60), "Hút", invisible if: PR_Line02.bCupSuctionValve, input disabled if: PR_Line02.bCupSuctionValve
        OnMouseDown: execute { PR_Line02.bCupSuctionValve := true; }
    Image (510,126 500x500), image: ImagePool.Cumcapnap
    Rectangle (5,505 350x50), "4. Van hút định vị hũ"
    Rectangle (5,115 350x50), "1. Ben hút, thả nắp"
    Rectangle (5,245 350x50), "2. Ben chặn nắp trên ray"
    Rectangle (5,375 350x50), "3. Van hút nắp"
    Frame (0,650 1024x35)
        shows N_Footer_Alarm()
END_VISUALIZATION

// ---- VISUs/Manual/Line2/N_Tranfer2.TcVIS
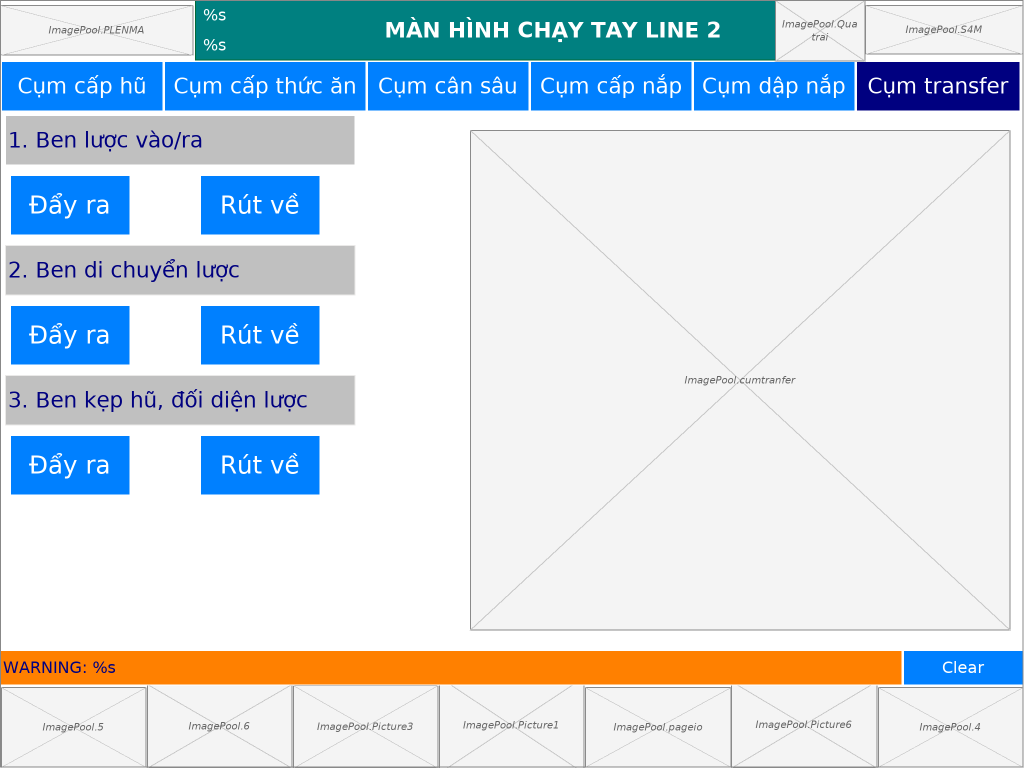
VISUALIZATION N_Tranfer2  // 1024x768
    Rectangle (10,305 120x60), "Đẩy ra", colour toggle: PR_Line02.bCylinder_Move_Comb_Extend, input disabled if: Not PR_Line02.bCheck
        OnMouseDown: execute { PR_Line02.bCylinder_Move_Comb_Extend := TRUE; PR_Line02.bCylinder_Move_Comb_Retract := FALSE; }
    Rectangle (200,175 120x60), "Rút về", colour toggle: PR_Line02.bCylinder_Comb_Retract
        OnMouseDown: execute { PR_Line02.bCylinder_Comb_Retract := TRUE; PR_Line02.bCylinder_Comb_Extend := FALSE; }
    Rectangle (200,305 120x60), "Rút về", colour toggle: PR_Line02.bCylinder_Move_Comb_Retract, input disabled if: Not PR_Line02.bCheck
        OnMouseDown: execute { PR_Line02.bCylinder_Move_Comb_Retract := TRUE; PR_Line02.bCylinder_Move_Comb_Extend := FALSE; }
    Frame (0,687 1024x80)
        shows N_Footer_Line2()
    Frame (0,0 1024x60)
        shows N_Header()
    Textfield (353,5 400x50), "MÀN HÌNH CHẠY TAY LINE 2"
    Rectangle (10,175 120x60), "Đẩy ra", colour toggle: PR_Line02.bCylinder_Comb_Extend, input disabled if: Not PR_Line02.bCheck
        OnMouseDown: execute { PR_Line02.bCylinder_Comb_Extend := TRUE; PR_Line02.bCylinder_Comb_Retract := FALSE; }
    Rectangle (1,61 162x50), "Cụm cấp hũ"
        OnMouseClick: change screen: N_JarSupply2
    Rectangle (164,61 202x50), "Cụm cấp thức ăn"
        OnMouseClick: change screen: N_FoodSupply2
    Rectangle (367,61 162x50), "Cụm cân sâu"
        OnMouseClick: change screen: N_WormWeight2
    Rectangle (530,61 162x50), "Cụm cấp nắp"
        OnMouseClick: change screen: N_LidSupply2
    Rectangle (693,61 162x50), "Cụm dập nắp"
        OnMouseClick: change screen: N_LidPressing2
    Rectangle (856,61 164x50), "Cụm transfer"
        OnMouseClick: change screen: N_Tranfer2
    Rectangle (200,435 120x60), "Rút về", colour toggle: PR_Line02.bCylinder_Clip_Retract
        OnMouseDown: execute { PR_Line02.bCylinder_Clip_Retract := TRUE; PR_Line02.bCylinder_Clip_Extend := FALSE; }
    Rectangle (10,435 120x60), "Đẩy ra", colour toggle: PR_Line02.bCylinder_Clip_Extend
        OnMouseDown: execute { PR_Line02.bCylinder_Clip_Extend := TRUE; PR_Line02.bCylinder_Clip_Retract := FALSE; }
    Image (775,0 90x61), input disabled if: bResetAuto1, image: ImagePool.Qua trai
        OnMouseClick: change screen: N_Tranfer1
        OnMouseClick: execute { MAIN.bModeManual := TRUE; MAIN.bModeAuto := FALSE; }
    Rectangle (5,115 350x50), "1. Ben lược vào/ra"
    Rectangle (5,245 350x50), "2. Ben di chuyển lược"
    Rectangle (5,375 350x50), "3. Ben kẹp hũ, đối diện lược"
    Image (470,130 540x500), image: ImagePool.cumtranfer
    Frame (0,650 1024x35)
        shows N_Footer_Alarm()
END_VISUALIZATION

// ---- VISUs/Manual/Line2/N_WormWeight2.TcVIS
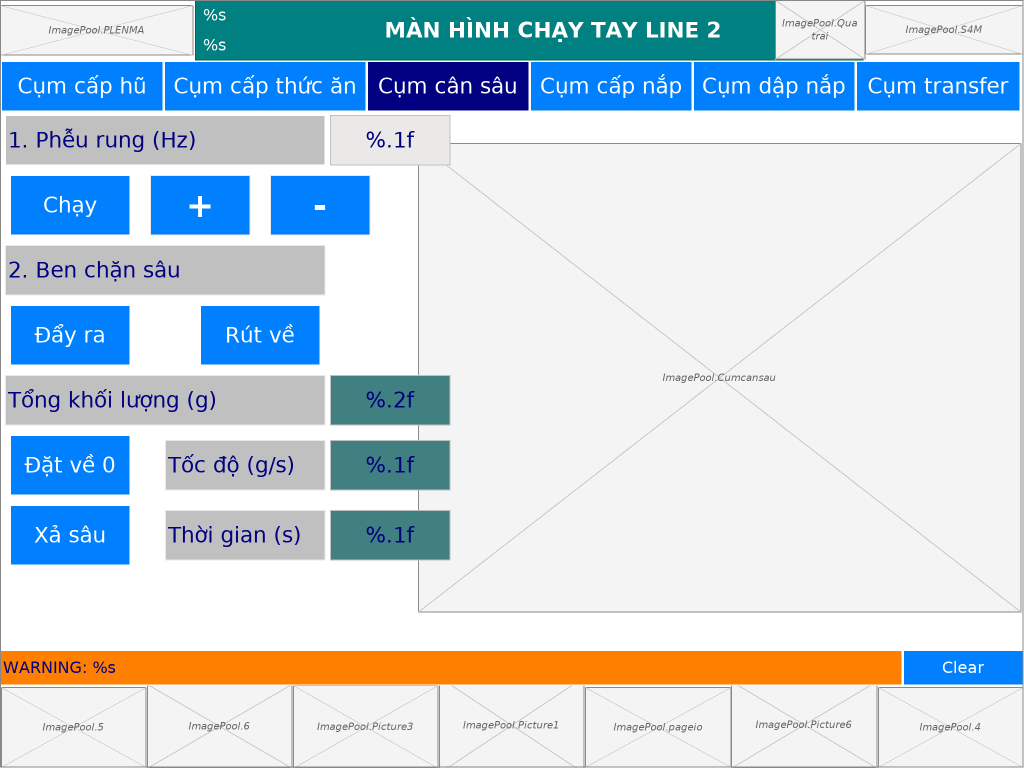
VISUALIZATION N_WormWeight2  // 1024x768
    Image (418,143 603x469), image: ImagePool.Cumcansau
    Rectangle (10,305 120x60), "Đẩy ra", colour toggle: PR_Line02.bCylinder_Block_Worm_Extend
        OnMouseDown: execute {
            PR_Line02.bCylinder_Block_Worm_Extend := TRUE;
            PR_Line02.bCylinder_Block_Worm_Retract := FALSE;
            PR_Line02.bxa := FALSE;
        }
    Rectangle (10,175 120x60), "Dừng", invisible if: not PR_Line02.bMotor_vibrating_funnel, input disabled if: not PR_Line02.bMotor_vibrating_funnel
        OnMouseDown: execute { PR_Line02.bMotor_vibrating_funnel := false; }
    Rectangle (200,305 120x60), "Rút về", colour toggle: PR_Line02.bCylinder_Block_Worm_Retract
        OnMouseDown: execute {
            PR_Line02.bCylinder_Block_Worm_Retract := TRUE;
            PR_Line02.bCylinder_Block_Worm_Extend := FALSE;
            PR_Line02.bxa := FALSE;
        }
    Frame (0,687 1024x80)
        shows N_Footer_Line2()
    Frame (0,0 1024x60)
        shows N_Header()
    Textfield (353,5 400x50), "MÀN HÌNH CHẠY TAY LINE 2"
    Rectangle (10,175 120x60), "Chạy", invisible if: PR_Line02.bMotor_vibrating_funnel, input disabled if: PR_Line02.bMotor_vibrating_funnel
        OnMouseDown: execute { PR_Line02.bMotor_vibrating_funnel := TRUE; PR_Line02.bxa := FALSE; }
    Rectangle (330,115 120x50), "%.1f", text variable: PR_Line02.fb_WormWeight.fSpeed_vibrating_funnel_Manual
        OnMouseDown: write PR_Line02.fb_WormWeight.fSpeed_vibrating_funnel_Manual via VisuDialogs.Numpad
        OnMouseDown: execute { PR_Line02.bxa := FALSE; }
    Rectangle (150,175 100x60), "+", colour toggle: PR_Line02.bUp_vibrating_funnel
        OnMouseDown: execute { PR_Line02.bUp_vibrating_funnel := TRUE; PR_Line02.bxa := FALSE; }
    Rectangle (270,175 100x60), "-", colour toggle: PR_Line02.bDown_vibrating_funnel
        OnMouseDown: execute { PR_Line02.bDown_vibrating_funnel := TRUE; PR_Line02.bxa := FALSE; }
    Rectangle (330,375 120x50), "%.2f", text variable: PR_Line02.fb_WormWeight.fWeight_Worm
    Rectangle (10,435 120x60), "Đặt về 0"
        tap PR_Line02.bZero_Loadcell_Worm
        OnMouseDown: execute { PR_Line02.bxa := FALSE; }
        OnMouseUp: execute { PR_Line02.bZero_Loadcell_Worm := TRUE; }
    Rectangle (330,440 120x50), "%.1f", text variable: PR_Line02.fb_WormWeight.fFlow_Worm
    Image (775,0 90x59), input disabled if: bResetAuto1, image: ImagePool.Qua trai
        OnMouseClick: change screen: N_WormWeight1
        OnMouseClick: execute { MAIN.bModeManual := TRUE; MAIN.bModeAuto := FALSE; }
    Rectangle (1,61 162x50), "Cụm cấp hũ"
        OnMouseClick: change screen: N_JarSupply2
    Rectangle (164,61 202x50), "Cụm cấp thức ăn"
        OnMouseClick: change screen: N_FoodSupply2
    Rectangle (367,61 162x50), "Cụm cân sâu"
        OnMouseClick: change screen: N_WormWeight2
    Rectangle (530,61 162x50), "Cụm cấp nắp"
        OnMouseClick: change screen: N_LidSupply2
    Rectangle (693,61 162x50), "Cụm dập nắp"
        OnMouseClick: change screen: N_LidPressing2
    Rectangle (856,61 164x50), "Cụm transfer"
        OnMouseClick: change screen: N_Tranfer2
    Rectangle (5,375 320x50), "Tổng khối lượng (g)"
    Rectangle (5,115 320x50), "1. Phễu rung (Hz)"
    Rectangle (5,245 320x50), "2. Ben chặn sâu"
    Rectangle (165,440 160x50), "Tốc độ (g/s)"
    Rectangle (165,510 160x50), "Thời gian (s)"
    Rectangle (10,505 120x60), "Xả sâu", colour toggle: PR_Line02.xasau
        OnMouseDown: execute { PR_Line02.xasau := TRUE; PR_Line02.bxa := true; }
    Rectangle (330,510 120x50), "%.1f", text variable: PR_Line02.fb_WormWeight.fTime
    Frame (0,650 1024x35)
        shows N_Footer_Alarm()
END_VISUALIZATION

// ---- VISUs/Recipe/N_Recipe_Line1.TcVIS
